	WY10200_00 AT  %MX10200.0 : BOOL; (*STN 5 PROCESS TANK HEATER A ON/OFF (-70K1) *)
	WY10200_01 AT  %MX10200.1 : BOOL; (*STN 5 PROCESS TANK HEATER A ON/OFF (-70K1) *)
	WY10200_02 AT  %MX10200.2 : BOOL; (*STN 5 PROCESS TANK HEATER A ON/OFF (-70K1) *)
	WY10200_03 AT  %MX10200.3 : BOOL; (*STN 5 PROCESS TANK HEATER A ON/OFF (-70K1) *)
	WY10200_04 AT  %MX10200.4 : BOOL; (*STN 5 PROCESS TANK HEATER A ON/OFF (-70K1) *)
	WY10200_05 AT  %MX10200.5 : BOOL; (*STN 5 PROCESS TANK HEATER A ON/OFF (-70K1) *)
	WY10200_06 AT  %MX10200.6 : BOOL; (*STN 5 PROCESS TANK HEATER A ON/OFF (-70K1) *)
	WY10200_07 AT  %MX10200.7 : BOOL; (*STN 5 PROCESS TANK HEATER A ON/OFF (-70K1) *)
	WY10200_08 AT  %MX10200.8 : BOOL; (*STN 5 PROCESS TANK HEATER A ON/OFF (-70K1) *)
	WY10200_09 AT  %MX10200.9 : BOOL; (*STN 5 PROCESS TANK HEATER A ON/OFF (-70K1) *)
	WY10200_10 AT  %MX10200.10 : BOOL; (*STN 5 PROCESS TANK HEATER A ON/OFF (-70K1) *)
	WY10200_11 AT  %MX10200.11 : BOOL; (*STN 5 PROCESS TANK HEATER A ON/OFF (-70K1) *)
	WY10200_12 AT  %MX10200.12 : BOOL; (*STN 5 PROCESS TANK HEATER A ON/OFF (-70K1) *)
	WY10200_13 AT  %MX10200.13 : BOOL; (*STN 5 PROCESS TANK HEATER A ON/OFF (-70K1) *)
	WY10200_14 AT  %MX10200.14 : BOOL; (*STN 5 PROCESS TANK HEATER A ON/OFF (-70K1) *)
	WY10200_15 AT  %MX10200.15 : BOOL; (*STN 5 PROCESS TANK HEATER A ON/OFF (-70K1) *)
	WY10200_16 AT  %MX10200.16 : BOOL; (*STN 5 PROCESS TANK HEATER A ON/OFF (-70K1) *)
	WY10200_17 AT  %MX10200.17 : BOOL; (*STN 5 PROCESS TANK HEATER A ON/OFF (-70K1) *)
	WY10200_18 AT  %MX10200.18 : BOOL; (*STN 5 PROCESS TANK HEATER A ON/OFF (-70K1) *)
	WY10200_19 AT  %MX10200.19 : BOOL; (*STN 5 PROCESS TANK HEATER A ON/OFF (-70K1) *)
	WY10200_20 AT  %MX10200.20 : BOOL; (*STN 5 PROCESS TANK HEATER A ON/OFF (-70K1) *)
	WY10200_21 AT  %MX10200.21 : BOOL; (*STN 5 PROCESS TANK HEATER A ON/OFF (-70K1) *)
	WY10200_22 AT  %MX10200.22 : BOOL; (*STN 5 PROCESS TANK HEATER A ON/OFF (-70K1) *)
	WY10200_23 AT  %MX10200.23 : BOOL; (*STN 5 PROCESS TANK HEATER A ON/OFF (-70K1) *)
	WY10200_24 AT  %MX10200.24 : BOOL; (*STN 5 PROCESS TANK HEATER A ON/OFF (-70K1) *)
	WY10200_25 AT  %MX10200.25 : BOOL; (*STN 5 PROCESS TANK HEATER A ON/OFF (-70K1) *)
	WY10200_26 AT  %MX10200.26 : BOOL; (*STN 5 PROCESS TANK HEATER A ON/OFF (-70K1) *)
	WY10200_27 AT  %MX10200.27 : BOOL; (*STN 5 PROCESS TANK HEATER A ON/OFF (-70K1) *)
	WY10200_28 AT  %MX10200.28 : BOOL; (*STN 5 PROCESS TANK HEATER A ON/OFF (-70K1) *)
	WY10200_29 AT  %MX10200.29 : BOOL; (*STN 5 PROCESS TANK HEATER A ON/OFF (-70K1) *)
	WY10200_30 AT  %MX10200.30 : BOOL; (*STN 5 PROCESS TANK HEATER A ON/OFF (-70K1) *)
	WY10200_31 AT  %MX10200.31 : BOOL; (*STN 5 PROCESS TANK HEATER A ON/OFF (-70K1) *)

	WY10201_00 AT  %MX10204.0 : BOOL; (*STN 5 PROCESS TANK HEATER B ON/OFF (-71K1) *)
	WY10201_01 AT  %MX10204.1 : BOOL; (*STN 5 PROCESS TANK HEATER B ON/OFF (-71K1) *)
	WY10201_02 AT  %MX10204.2 : BOOL; (*STN 5 PROCESS TANK HEATER B ON/OFF (-71K1) *)
	WY10201_03 AT  %MX10204.3 : BOOL; (*STN 5 PROCESS TANK HEATER B ON/OFF (-71K1) *)
	WY10201_04 AT  %MX10204.4 : BOOL; (*STN 5 PROCESS TANK HEATER B ON/OFF (-71K1) *)
	WY10201_05 AT  %MX10204.5 : BOOL; (*STN 5 PROCESS TANK HEATER B ON/OFF (-71K1) *)
	WY10201_06 AT  %MX10204.6 : BOOL; (*STN 5 PROCESS TANK HEATER B ON/OFF (-71K1) *)
	WY10201_07 AT  %MX10204.7 : BOOL; (*STN 5 PROCESS TANK HEATER B ON/OFF (-71K1) *)
	WY10201_08 AT  %MX10204.8 : BOOL; (*STN 5 PROCESS TANK HEATER B ON/OFF (-71K1) *)
	WY10201_09 AT  %MX10204.9 : BOOL; (*STN 5 PROCESS TANK HEATER B ON/OFF (-71K1) *)
	WY10201_10 AT  %MX10204.10 : BOOL; (*STN 5 PROCESS TANK HEATER B ON/OFF (-71K1) *)
	WY10201_11 AT  %MX10204.11 : BOOL; (*STN 5 PROCESS TANK HEATER B ON/OFF (-71K1) *)
	WY10201_12 AT  %MX10204.12 : BOOL; (*STN 5 PROCESS TANK HEATER B ON/OFF (-71K1) *)
	WY10201_13 AT  %MX10204.13 : BOOL; (*STN 5 PROCESS TANK HEATER B ON/OFF (-71K1) *)
	WY10201_14 AT  %MX10204.14 : BOOL; (*STN 5 PROCESS TANK HEATER B ON/OFF (-71K1) *)
	WY10201_15 AT  %MX10204.15 : BOOL; (*STN 5 PROCESS TANK HEATER B ON/OFF (-71K1) *)
	WY10201_16 AT  %MX10204.16 : BOOL; (*STN 5 PROCESS TANK HEATER B ON/OFF (-71K1) *)
	WY10201_17 AT  %MX10204.17 : BOOL; (*STN 5 PROCESS TANK HEATER B ON/OFF (-71K1) *)
	WY10201_18 AT  %MX10204.18 : BOOL; (*STN 5 PROCESS TANK HEATER B ON/OFF (-71K1) *)
	WY10201_19 AT  %MX10204.19 : BOOL; (*STN 5 PROCESS TANK HEATER B ON/OFF (-71K1) *)
	WY10201_20 AT  %MX10204.20 : BOOL; (*STN 5 PROCESS TANK HEATER B ON/OFF (-71K1) *)
	WY10201_21 AT  %MX10204.21 : BOOL; (*STN 5 PROCESS TANK HEATER B ON/OFF (-71K1) *)
	WY10201_22 AT  %MX10204.22 : BOOL; (*STN 5 PROCESS TANK HEATER B ON/OFF (-71K1) *)
	WY10201_23 AT  %MX10204.23 : BOOL; (*STN 5 PROCESS TANK HEATER B ON/OFF (-71K1) *)
	WY10201_24 AT  %MX10204.24 : BOOL; (*STN 5 PROCESS TANK HEATER B ON/OFF (-71K1) *)
	WY10201_25 AT  %MX10204.25 : BOOL; (*STN 5 PROCESS TANK HEATER B ON/OFF (-71K1) *)
	WY10201_26 AT  %MX10204.26 : BOOL; (*STN 5 PROCESS TANK HEATER B ON/OFF (-71K1) *)
	WY10201_27 AT  %MX10204.27 : BOOL; (*STN 5 PROCESS TANK HEATER B ON/OFF (-71K1) *)
	WY10201_28 AT  %MX10204.28 : BOOL; (*STN 5 PROCESS TANK HEATER B ON/OFF (-71K1) *)
	WY10201_29 AT  %MX10204.29 : BOOL; (*STN 5 PROCESS TANK HEATER B ON/OFF (-71K1) *)
	WY10201_30 AT  %MX10204.30 : BOOL; (*STN 5 PROCESS TANK HEATER B ON/OFF (-71K1) *)
	WY10201_31 AT  %MX10204.31 : BOOL; (*STN 5 PROCESS TANK HEATER B ON/OFF (-71K1) *)

	WY10202_00 AT  %MX10208.0 : BOOL; (*STN 1 SUB PROCESS TANK HEATER ON/OFF (-72K1) *)
	WY10202_01 AT  %MX10208.1 : BOOL; (*STN 1 SUB PROCESS TANK HEATER ON/OFF (-72K1) *)
	WY10202_02 AT  %MX10208.2 : BOOL; (*STN 1 SUB PROCESS TANK HEATER ON/OFF (-72K1) *)
	WY10202_03 AT  %MX10208.3 : BOOL; (*STN 1 SUB PROCESS TANK HEATER ON/OFF (-72K1) *)
	WY10202_04 AT  %MX10208.4 : BOOL; (*STN 1 SUB PROCESS TANK HEATER ON/OFF (-72K1) *)
	WY10202_05 AT  %MX10208.5 : BOOL; (*STN 1 SUB PROCESS TANK HEATER ON/OFF (-72K1) *)
	WY10202_06 AT  %MX10208.6 : BOOL; (*STN 1 SUB PROCESS TANK HEATER ON/OFF (-72K1) *)
	WY10202_07 AT  %MX10208.7 : BOOL; (*STN 1 SUB PROCESS TANK HEATER ON/OFF (-72K1) *)
	WY10202_08 AT  %MX10208.8 : BOOL; (*STN 1 SUB PROCESS TANK HEATER ON/OFF (-72K1) *)
	WY10202_09 AT  %MX10208.9 : BOOL; (*STN 1 SUB PROCESS TANK HEATER ON/OFF (-72K1) *)
	WY10202_10 AT  %MX10208.10 : BOOL; (*STN 1 SUB PROCESS TANK HEATER ON/OFF (-72K1) *)
	WY10202_11 AT  %MX10208.11 : BOOL; (*STN 1 SUB PROCESS TANK HEATER ON/OFF (-72K1) *)
	WY10202_12 AT  %MX10208.12 : BOOL; (*STN 1 SUB PROCESS TANK HEATER ON/OFF (-72K1) *)
	WY10202_13 AT  %MX10208.13 : BOOL; (*STN 1 SUB PROCESS TANK HEATER ON/OFF (-72K1) *)
	WY10202_14 AT  %MX10208.14 : BOOL; (*STN 1 SUB PROCESS TANK HEATER ON/OFF (-72K1) *)
	WY10202_15 AT  %MX10208.15 : BOOL; (*STN 1 SUB PROCESS TANK HEATER ON/OFF (-72K1) *)
	WY10202_16 AT  %MX10208.16 : BOOL; (*STN 1 SUB PROCESS TANK HEATER ON/OFF (-72K1) *)
	WY10202_17 AT  %MX10208.17 : BOOL; (*STN 1 SUB PROCESS TANK HEATER ON/OFF (-72K1) *)
	WY10202_18 AT  %MX10208.18 : BOOL; (*STN 1 SUB PROCESS TANK HEATER ON/OFF (-72K1) *)
	WY10202_19 AT  %MX10208.19 : BOOL; (*STN 1 SUB PROCESS TANK HEATER ON/OFF (-72K1) *)
	WY10202_20 AT  %MX10208.20 : BOOL; (*STN 1 SUB PROCESS TANK HEATER ON/OFF (-72K1) *)
	WY10202_21 AT  %MX10208.21 : BOOL; (*STN 1 SUB PROCESS TANK HEATER ON/OFF (-72K1) *)
	WY10202_22 AT  %MX10208.22 : BOOL; (*STN 1 SUB PROCESS TANK HEATER ON/OFF (-72K1) *)
	WY10202_23 AT  %MX10208.23 : BOOL; (*STN 1 SUB PROCESS TANK HEATER ON/OFF (-72K1) *)
	WY10202_24 AT  %MX10208.24 : BOOL; (*STN 1 SUB PROCESS TANK HEATER ON/OFF (-72K1) *)
	WY10202_25 AT  %MX10208.25 : BOOL; (*STN 1 SUB PROCESS TANK HEATER ON/OFF (-72K1) *)
	WY10202_26 AT  %MX10208.26 : BOOL; (*STN 1 SUB PROCESS TANK HEATER ON/OFF (-72K1) *)
	WY10202_27 AT  %MX10208.27 : BOOL; (*STN 1 SUB PROCESS TANK HEATER ON/OFF (-72K1) *)
	WY10202_28 AT  %MX10208.28 : BOOL; (*STN 1 SUB PROCESS TANK HEATER ON/OFF (-72K1) *)
	WY10202_29 AT  %MX10208.29 : BOOL; (*STN 1 SUB PROCESS TANK HEATER ON/OFF (-72K1) *)
	WY10202_30 AT  %MX10208.30 : BOOL; (*STN 1 SUB PROCESS TANK HEATER ON/OFF (-72K1) *)
	WY10202_31 AT  %MX10208.31 : BOOL; (*STN 1 SUB PROCESS TANK HEATER ON/OFF (-72K1) *)

	WY10203_00 AT  %MX10212.0 : BOOL; (*STN 2 SUB PROCESS TANK HEATER ON/OFF (-73K1) *)
	WY10203_01 AT  %MX10212.1 : BOOL; (*STN 2 SUB PROCESS TANK HEATER ON/OFF (-73K1) *)
	WY10203_02 AT  %MX10212.2 : BOOL; (*STN 2 SUB PROCESS TANK HEATER ON/OFF (-73K1) *)
	WY10203_03 AT  %MX10212.3 : BOOL; (*STN 2 SUB PROCESS TANK HEATER ON/OFF (-73K1) *)
	WY10203_04 AT  %MX10212.4 : BOOL; (*STN 2 SUB PROCESS TANK HEATER ON/OFF (-73K1) *)
	WY10203_05 AT  %MX10212.5 : BOOL; (*STN 2 SUB PROCESS TANK HEATER ON/OFF (-73K1) *)
	WY10203_06 AT  %MX10212.6 : BOOL; (*STN 2 SUB PROCESS TANK HEATER ON/OFF (-73K1) *)
	WY10203_07 AT  %MX10212.7 : BOOL; (*STN 2 SUB PROCESS TANK HEATER ON/OFF (-73K1) *)
	WY10203_08 AT  %MX10212.8 : BOOL; (*STN 2 SUB PROCESS TANK HEATER ON/OFF (-73K1) *)
	WY10203_09 AT  %MX10212.9 : BOOL; (*STN 2 SUB PROCESS TANK HEATER ON/OFF (-73K1) *)
	WY10203_10 AT  %MX10212.10 : BOOL; (*STN 2 SUB PROCESS TANK HEATER ON/OFF (-73K1) *)
	WY10203_11 AT  %MX10212.11 : BOOL; (*STN 2 SUB PROCESS TANK HEATER ON/OFF (-73K1) *)
	WY10203_12 AT  %MX10212.12 : BOOL; (*STN 2 SUB PROCESS TANK HEATER ON/OFF (-73K1) *)
	WY10203_13 AT  %MX10212.13 : BOOL; (*STN 2 SUB PROCESS TANK HEATER ON/OFF (-73K1) *)
	WY10203_14 AT  %MX10212.14 : BOOL; (*STN 2 SUB PROCESS TANK HEATER ON/OFF (-73K1) *)
	WY10203_15 AT  %MX10212.15 : BOOL; (*STN 2 SUB PROCESS TANK HEATER ON/OFF (-73K1) *)
	WY10203_16 AT  %MX10212.16 : BOOL; (*STN 2 SUB PROCESS TANK HEATER ON/OFF (-73K1) *)
	WY10203_17 AT  %MX10212.17 : BOOL; (*STN 2 SUB PROCESS TANK HEATER ON/OFF (-73K1) *)
	WY10203_18 AT  %MX10212.18 : BOOL; (*STN 2 SUB PROCESS TANK HEATER ON/OFF (-73K1) *)
	WY10203_19 AT  %MX10212.19 : BOOL; (*STN 2 SUB PROCESS TANK HEATER ON/OFF (-73K1) *)
	WY10203_20 AT  %MX10212.20 : BOOL; (*STN 2 SUB PROCESS TANK HEATER ON/OFF (-73K1) *)
	WY10203_21 AT  %MX10212.21 : BOOL; (*STN 2 SUB PROCESS TANK HEATER ON/OFF (-73K1) *)
	WY10203_22 AT  %MX10212.22 : BOOL; (*STN 2 SUB PROCESS TANK HEATER ON/OFF (-73K1) *)
	WY10203_23 AT  %MX10212.23 : BOOL; (*STN 2 SUB PROCESS TANK HEATER ON/OFF (-73K1) *)
	WY10203_24 AT  %MX10212.24 : BOOL; (*STN 2 SUB PROCESS TANK HEATER ON/OFF (-73K1) *)
	WY10203_25 AT  %MX10212.25 : BOOL; (*STN 2 SUB PROCESS TANK HEATER ON/OFF (-73K1) *)
	WY10203_26 AT  %MX10212.26 : BOOL; (*STN 2 SUB PROCESS TANK HEATER ON/OFF (-73K1) *)
	WY10203_27 AT  %MX10212.27 : BOOL; (*STN 2 SUB PROCESS TANK HEATER ON/OFF (-73K1) *)
	WY10203_28 AT  %MX10212.28 : BOOL; (*STN 2 SUB PROCESS TANK HEATER ON/OFF (-73K1) *)
	WY10203_29 AT  %MX10212.29 : BOOL; (*STN 2 SUB PROCESS TANK HEATER ON/OFF (-73K1) *)
	WY10203_30 AT  %MX10212.30 : BOOL; (*STN 2 SUB PROCESS TANK HEATER ON/OFF (-73K1) *)
	WY10203_31 AT  %MX10212.31 : BOOL; (*STN 2 SUB PROCESS TANK HEATER ON/OFF (-73K1) *)

	WY10204_00 AT  %MX10216.0 : BOOL; (*STN 3 SUB PROCESS TANK HEATER ON/OFF (-74K1) *)
	WY10204_01 AT  %MX10216.1 : BOOL; (*STN 3 SUB PROCESS TANK HEATER ON/OFF (-74K1) *)
	WY10204_02 AT  %MX10216.2 : BOOL; (*STN 3 SUB PROCESS TANK HEATER ON/OFF (-74K1) *)
	WY10204_03 AT  %MX10216.3 : BOOL; (*STN 3 SUB PROCESS TANK HEATER ON/OFF (-74K1) *)
	WY10204_04 AT  %MX10216.4 : BOOL; (*STN 3 SUB PROCESS TANK HEATER ON/OFF (-74K1) *)
	WY10204_05 AT  %MX10216.5 : BOOL; (*STN 3 SUB PROCESS TANK HEATER ON/OFF (-74K1) *)
	WY10204_06 AT  %MX10216.6 : BOOL; (*STN 3 SUB PROCESS TANK HEATER ON/OFF (-74K1) *)
	WY10204_07 AT  %MX10216.7 : BOOL; (*STN 3 SUB PROCESS TANK HEATER ON/OFF (-74K1) *)
	WY10204_08 AT  %MX10216.8 : BOOL; (*STN 3 SUB PROCESS TANK HEATER ON/OFF (-74K1) *)
	WY10204_09 AT  %MX10216.9 : BOOL; (*STN 3 SUB PROCESS TANK HEATER ON/OFF (-74K1) *)
	WY10204_10 AT  %MX10216.10 : BOOL; (*STN 3 SUB PROCESS TANK HEATER ON/OFF (-74K1) *)
	WY10204_11 AT  %MX10216.11 : BOOL; (*STN 3 SUB PROCESS TANK HEATER ON/OFF (-74K1) *)
	WY10204_12 AT  %MX10216.12 : BOOL; (*STN 3 SUB PROCESS TANK HEATER ON/OFF (-74K1) *)
	WY10204_13 AT  %MX10216.13 : BOOL; (*STN 3 SUB PROCESS TANK HEATER ON/OFF (-74K1) *)
	WY10204_14 AT  %MX10216.14 : BOOL; (*STN 3 SUB PROCESS TANK HEATER ON/OFF (-74K1) *)
	WY10204_15 AT  %MX10216.15 : BOOL; (*STN 3 SUB PROCESS TANK HEATER ON/OFF (-74K1) *)
	WY10204_16 AT  %MX10216.16 : BOOL; (*STN 3 SUB PROCESS TANK HEATER ON/OFF (-74K1) *)
	WY10204_17 AT  %MX10216.17 : BOOL; (*STN 3 SUB PROCESS TANK HEATER ON/OFF (-74K1) *)
	WY10204_18 AT  %MX10216.18 : BOOL; (*STN 3 SUB PROCESS TANK HEATER ON/OFF (-74K1) *)
	WY10204_19 AT  %MX10216.19 : BOOL; (*STN 3 SUB PROCESS TANK HEATER ON/OFF (-74K1) *)
	WY10204_20 AT  %MX10216.20 : BOOL; (*STN 3 SUB PROCESS TANK HEATER ON/OFF (-74K1) *)
	WY10204_21 AT  %MX10216.21 : BOOL; (*STN 3 SUB PROCESS TANK HEATER ON/OFF (-74K1) *)
	WY10204_22 AT  %MX10216.22 : BOOL; (*STN 3 SUB PROCESS TANK HEATER ON/OFF (-74K1) *)
	WY10204_23 AT  %MX10216.23 : BOOL; (*STN 3 SUB PROCESS TANK HEATER ON/OFF (-74K1) *)
	WY10204_24 AT  %MX10216.24 : BOOL; (*STN 3 SUB PROCESS TANK HEATER ON/OFF (-74K1) *)
	WY10204_25 AT  %MX10216.25 : BOOL; (*STN 3 SUB PROCESS TANK HEATER ON/OFF (-74K1) *)
	WY10204_26 AT  %MX10216.26 : BOOL; (*STN 3 SUB PROCESS TANK HEATER ON/OFF (-74K1) *)
	WY10204_27 AT  %MX10216.27 : BOOL; (*STN 3 SUB PROCESS TANK HEATER ON/OFF (-74K1) *)
	WY10204_28 AT  %MX10216.28 : BOOL; (*STN 3 SUB PROCESS TANK HEATER ON/OFF (-74K1) *)
	WY10204_29 AT  %MX10216.29 : BOOL; (*STN 3 SUB PROCESS TANK HEATER ON/OFF (-74K1) *)
	WY10204_30 AT  %MX10216.30 : BOOL; (*STN 3 SUB PROCESS TANK HEATER ON/OFF (-74K1) *)
	WY10204_31 AT  %MX10216.31 : BOOL; (*STN 3 SUB PROCESS TANK HEATER ON/OFF (-74K1) *)

	WY10205_00 AT  %MX10220.0 : BOOL; (*MAIN INC HEATER ON/OFF   (-75K1) *)
	WY10205_01 AT  %MX10220.1 : BOOL; (*MAIN INC HEATER ON/OFF   (-75K1) *)
	WY10205_02 AT  %MX10220.2 : BOOL; (*MAIN INC HEATER ON/OFF   (-75K1) *)
	WY10205_03 AT  %MX10220.3 : BOOL; (*MAIN INC HEATER ON/OFF   (-75K1) *)
	WY10205_04 AT  %MX10220.4 : BOOL; (*MAIN INC HEATER ON/OFF   (-75K1) *)
	WY10205_05 AT  %MX10220.5 : BOOL; (*MAIN INC HEATER ON/OFF   (-75K1) *)
	WY10205_06 AT  %MX10220.6 : BOOL; (*MAIN INC HEATER ON/OFF   (-75K1) *)
	WY10205_07 AT  %MX10220.7 : BOOL; (*MAIN INC HEATER ON/OFF   (-75K1) *)
	WY10205_08 AT  %MX10220.8 : BOOL; (*MAIN INC HEATER ON/OFF   (-75K1) *)
	WY10205_09 AT  %MX10220.9 : BOOL; (*MAIN INC HEATER ON/OFF   (-75K1) *)
	WY10205_10 AT  %MX10220.10 : BOOL; (*MAIN INC HEATER ON/OFF   (-75K1) *)
	WY10205_11 AT  %MX10220.11 : BOOL; (*MAIN INC HEATER ON/OFF   (-75K1) *)
	WY10205_12 AT  %MX10220.12 : BOOL; (*MAIN INC HEATER ON/OFF   (-75K1) *)
	WY10205_13 AT  %MX10220.13 : BOOL; (*MAIN INC HEATER ON/OFF   (-75K1) *)
	WY10205_14 AT  %MX10220.14 : BOOL; (*MAIN INC HEATER ON/OFF   (-75K1) *)
	WY10205_15 AT  %MX10220.15 : BOOL; (*MAIN INC HEATER ON/OFF   (-75K1) *)
	WY10205_16 AT  %MX10220.16 : BOOL; (*MAIN INC HEATER ON/OFF   (-75K1) *)
	WY10205_17 AT  %MX10220.17 : BOOL; (*MAIN INC HEATER ON/OFF   (-75K1) *)
	WY10205_18 AT  %MX10220.18 : BOOL; (*MAIN INC HEATER ON/OFF   (-75K1) *)
	WY10205_19 AT  %MX10220.19 : BOOL; (*MAIN INC HEATER ON/OFF   (-75K1) *)
	WY10205_20 AT  %MX10220.20 : BOOL; (*MAIN INC HEATER ON/OFF   (-75K1) *)
	WY10205_21 AT  %MX10220.21 : BOOL; (*MAIN INC HEATER ON/OFF   (-75K1) *)
	WY10205_22 AT  %MX10220.22 : BOOL; (*MAIN INC HEATER ON/OFF   (-75K1) *)
	WY10205_23 AT  %MX10220.23 : BOOL; (*MAIN INC HEATER ON/OFF   (-75K1) *)
	WY10205_24 AT  %MX10220.24 : BOOL; (*MAIN INC HEATER ON/OFF   (-75K1) *)
	WY10205_25 AT  %MX10220.25 : BOOL; (*MAIN INC HEATER ON/OFF   (-75K1) *)
	WY10205_26 AT  %MX10220.26 : BOOL; (*MAIN INC HEATER ON/OFF   (-75K1) *)
	WY10205_27 AT  %MX10220.27 : BOOL; (*MAIN INC HEATER ON/OFF   (-75K1) *)
	WY10205_28 AT  %MX10220.28 : BOOL; (*MAIN INC HEATER ON/OFF   (-75K1) *)
	WY10205_29 AT  %MX10220.29 : BOOL; (*MAIN INC HEATER ON/OFF   (-75K1) *)
	WY10205_30 AT  %MX10220.30 : BOOL; (*MAIN INC HEATER ON/OFF   (-75K1) *)
	WY10205_31 AT  %MX10220.31 : BOOL; (*MAIN INC HEATER ON/OFF   (-75K1) *)

	WY10206_00 AT  %MX10224.0 : BOOL; (*STN 1 ULTRASONIC FREQ ON/OFF (-16U1) *)
	WY10206_01 AT  %MX10224.1 : BOOL; (*STN 1 ULTRASONIC FREQ ON/OFF (-16U1) *)
	WY10206_02 AT  %MX10224.2 : BOOL; (*STN 1 ULTRASONIC FREQ ON/OFF (-16U1) *)
	WY10206_03 AT  %MX10224.3 : BOOL; (*STN 1 ULTRASONIC FREQ ON/OFF (-16U1) *)
	WY10206_04 AT  %MX10224.4 : BOOL; (*STN 1 ULTRASONIC FREQ ON/OFF (-16U1) *)
	WY10206_05 AT  %MX10224.5 : BOOL; (*STN 1 ULTRASONIC FREQ ON/OFF (-16U1) *)
	WY10206_06 AT  %MX10224.6 : BOOL; (*STN 1 ULTRASONIC FREQ ON/OFF (-16U1) *)
	WY10206_07 AT  %MX10224.7 : BOOL; (*STN 1 ULTRASONIC FREQ ON/OFF (-16U1) *)
	WY10206_08 AT  %MX10224.8 : BOOL; (*STN 1 ULTRASONIC FREQ ON/OFF (-16U1) *)
	WY10206_09 AT  %MX10224.9 : BOOL; (*STN 1 ULTRASONIC FREQ ON/OFF (-16U1) *)
	WY10206_10 AT  %MX10224.10 : BOOL; (*STN 1 ULTRASONIC FREQ ON/OFF (-16U1) *)
	WY10206_11 AT  %MX10224.11 : BOOL; (*STN 1 ULTRASONIC FREQ ON/OFF (-16U1) *)
	WY10206_12 AT  %MX10224.12 : BOOL; (*STN 1 ULTRASONIC FREQ ON/OFF (-16U1) *)
	WY10206_13 AT  %MX10224.13 : BOOL; (*STN 1 ULTRASONIC FREQ ON/OFF (-16U1) *)
	WY10206_14 AT  %MX10224.14 : BOOL; (*STN 1 ULTRASONIC FREQ ON/OFF (-16U1) *)
	WY10206_15 AT  %MX10224.15 : BOOL; (*STN 1 ULTRASONIC FREQ ON/OFF (-16U1) *)
	WY10206_16 AT  %MX10224.16 : BOOL; (*STN 1 ULTRASONIC FREQ ON/OFF (-16U1) *)
	WY10206_17 AT  %MX10224.17 : BOOL; (*STN 1 ULTRASONIC FREQ ON/OFF (-16U1) *)
	WY10206_18 AT  %MX10224.18 : BOOL; (*STN 1 ULTRASONIC FREQ ON/OFF (-16U1) *)
	WY10206_19 AT  %MX10224.19 : BOOL; (*STN 1 ULTRASONIC FREQ ON/OFF (-16U1) *)
	WY10206_20 AT  %MX10224.20 : BOOL; (*STN 1 ULTRASONIC FREQ ON/OFF (-16U1) *)
	WY10206_21 AT  %MX10224.21 : BOOL; (*STN 1 ULTRASONIC FREQ ON/OFF (-16U1) *)
	WY10206_22 AT  %MX10224.22 : BOOL; (*STN 1 ULTRASONIC FREQ ON/OFF (-16U1) *)
	WY10206_23 AT  %MX10224.23 : BOOL; (*STN 1 ULTRASONIC FREQ ON/OFF (-16U1) *)
	WY10206_24 AT  %MX10224.24 : BOOL; (*STN 1 ULTRASONIC FREQ ON/OFF (-16U1) *)
	WY10206_25 AT  %MX10224.25 : BOOL; (*STN 1 ULTRASONIC FREQ ON/OFF (-16U1) *)
	WY10206_26 AT  %MX10224.26 : BOOL; (*STN 1 ULTRASONIC FREQ ON/OFF (-16U1) *)
	WY10206_27 AT  %MX10224.27 : BOOL; (*STN 1 ULTRASONIC FREQ ON/OFF (-16U1) *)
	WY10206_28 AT  %MX10224.28 : BOOL; (*STN 1 ULTRASONIC FREQ ON/OFF (-16U1) *)
	WY10206_29 AT  %MX10224.29 : BOOL; (*STN 1 ULTRASONIC FREQ ON/OFF (-16U1) *)
	WY10206_30 AT  %MX10224.30 : BOOL; (*STN 1 ULTRASONIC FREQ ON/OFF (-16U1) *)
	WY10206_31 AT  %MX10224.31 : BOOL; (*STN 1 ULTRASONIC FREQ ON/OFF (-16U1) *)

	WY10207_00 AT  %MX10228.0 : BOOL; (*STN 2 ULTRASONIC FREQ ON/OFF (-17U1) *)
	WY10207_01 AT  %MX10228.1 : BOOL; (*STN 2 ULTRASONIC FREQ ON/OFF (-17U1) *)
	WY10207_02 AT  %MX10228.2 : BOOL; (*STN 2 ULTRASONIC FREQ ON/OFF (-17U1) *)
	WY10207_03 AT  %MX10228.3 : BOOL; (*STN 2 ULTRASONIC FREQ ON/OFF (-17U1) *)
	WY10207_04 AT  %MX10228.4 : BOOL; (*STN 2 ULTRASONIC FREQ ON/OFF (-17U1) *)
	WY10207_05 AT  %MX10228.5 : BOOL; (*STN 2 ULTRASONIC FREQ ON/OFF (-17U1) *)
	WY10207_06 AT  %MX10228.6 : BOOL; (*STN 2 ULTRASONIC FREQ ON/OFF (-17U1) *)
	WY10207_07 AT  %MX10228.7 : BOOL; (*STN 2 ULTRASONIC FREQ ON/OFF (-17U1) *)
	WY10207_08 AT  %MX10228.8 : BOOL; (*STN 2 ULTRASONIC FREQ ON/OFF (-17U1) *)
	WY10207_09 AT  %MX10228.9 : BOOL; (*STN 2 ULTRASONIC FREQ ON/OFF (-17U1) *)
	WY10207_10 AT  %MX10228.10 : BOOL; (*STN 2 ULTRASONIC FREQ ON/OFF (-17U1) *)
	WY10207_11 AT  %MX10228.11 : BOOL; (*STN 2 ULTRASONIC FREQ ON/OFF (-17U1) *)
	WY10207_12 AT  %MX10228.12 : BOOL; (*STN 2 ULTRASONIC FREQ ON/OFF (-17U1) *)
	WY10207_13 AT  %MX10228.13 : BOOL; (*STN 2 ULTRASONIC FREQ ON/OFF (-17U1) *)
	WY10207_14 AT  %MX10228.14 : BOOL; (*STN 2 ULTRASONIC FREQ ON/OFF (-17U1) *)
	WY10207_15 AT  %MX10228.15 : BOOL; (*STN 2 ULTRASONIC FREQ ON/OFF (-17U1) *)
	WY10207_16 AT  %MX10228.16 : BOOL; (*STN 2 ULTRASONIC FREQ ON/OFF (-17U1) *)
	WY10207_17 AT  %MX10228.17 : BOOL; (*STN 2 ULTRASONIC FREQ ON/OFF (-17U1) *)
	WY10207_18 AT  %MX10228.18 : BOOL; (*STN 2 ULTRASONIC FREQ ON/OFF (-17U1) *)
	WY10207_19 AT  %MX10228.19 : BOOL; (*STN 2 ULTRASONIC FREQ ON/OFF (-17U1) *)
	WY10207_20 AT  %MX10228.20 : BOOL; (*STN 2 ULTRASONIC FREQ ON/OFF (-17U1) *)
	WY10207_21 AT  %MX10228.21 : BOOL; (*STN 2 ULTRASONIC FREQ ON/OFF (-17U1) *)
	WY10207_22 AT  %MX10228.22 : BOOL; (*STN 2 ULTRASONIC FREQ ON/OFF (-17U1) *)
	WY10207_23 AT  %MX10228.23 : BOOL; (*STN 2 ULTRASONIC FREQ ON/OFF (-17U1) *)
	WY10207_24 AT  %MX10228.24 : BOOL; (*STN 2 ULTRASONIC FREQ ON/OFF (-17U1) *)
	WY10207_25 AT  %MX10228.25 : BOOL; (*STN 2 ULTRASONIC FREQ ON/OFF (-17U1) *)
	WY10207_26 AT  %MX10228.26 : BOOL; (*STN 2 ULTRASONIC FREQ ON/OFF (-17U1) *)
	WY10207_27 AT  %MX10228.27 : BOOL; (*STN 2 ULTRASONIC FREQ ON/OFF (-17U1) *)
	WY10207_28 AT  %MX10228.28 : BOOL; (*STN 2 ULTRASONIC FREQ ON/OFF (-17U1) *)
	WY10207_29 AT  %MX10228.29 : BOOL; (*STN 2 ULTRASONIC FREQ ON/OFF (-17U1) *)
	WY10207_30 AT  %MX10228.30 : BOOL; (*STN 2 ULTRASONIC FREQ ON/OFF (-17U1) *)
	WY10207_31 AT  %MX10228.31 : BOOL; (*STN 2 ULTRASONIC FREQ ON/OFF (-17U1) *)

	WY10208_00 AT  %MX10232.0 : BOOL; (*STN 3 ULTRASONIC FREQ ON/OFF (-18U1) *)
	WY10208_01 AT  %MX10232.1 : BOOL; (*STN 3 ULTRASONIC FREQ ON/OFF (-18U1) *)
	WY10208_02 AT  %MX10232.2 : BOOL; (*STN 3 ULTRASONIC FREQ ON/OFF (-18U1) *)
	WY10208_03 AT  %MX10232.3 : BOOL; (*STN 3 ULTRASONIC FREQ ON/OFF (-18U1) *)
	WY10208_04 AT  %MX10232.4 : BOOL; (*STN 3 ULTRASONIC FREQ ON/OFF (-18U1) *)
	WY10208_05 AT  %MX10232.5 : BOOL; (*STN 3 ULTRASONIC FREQ ON/OFF (-18U1) *)
	WY10208_06 AT  %MX10232.6 : BOOL; (*STN 3 ULTRASONIC FREQ ON/OFF (-18U1) *)
	WY10208_07 AT  %MX10232.7 : BOOL; (*STN 3 ULTRASONIC FREQ ON/OFF (-18U1) *)
	WY10208_08 AT  %MX10232.8 : BOOL; (*STN 3 ULTRASONIC FREQ ON/OFF (-18U1) *)
	WY10208_09 AT  %MX10232.9 : BOOL; (*STN 3 ULTRASONIC FREQ ON/OFF (-18U1) *)
	WY10208_10 AT  %MX10232.10 : BOOL; (*STN 3 ULTRASONIC FREQ ON/OFF (-18U1) *)
	WY10208_11 AT  %MX10232.11 : BOOL; (*STN 3 ULTRASONIC FREQ ON/OFF (-18U1) *)
	WY10208_12 AT  %MX10232.12 : BOOL; (*STN 3 ULTRASONIC FREQ ON/OFF (-18U1) *)
	WY10208_13 AT  %MX10232.13 : BOOL; (*STN 3 ULTRASONIC FREQ ON/OFF (-18U1) *)
	WY10208_14 AT  %MX10232.14 : BOOL; (*STN 3 ULTRASONIC FREQ ON/OFF (-18U1) *)
	WY10208_15 AT  %MX10232.15 : BOOL; (*STN 3 ULTRASONIC FREQ ON/OFF (-18U1) *)
	WY10208_16 AT  %MX10232.16 : BOOL; (*STN 3 ULTRASONIC FREQ ON/OFF (-18U1) *)
	WY10208_17 AT  %MX10232.17 : BOOL; (*STN 3 ULTRASONIC FREQ ON/OFF (-18U1) *)
	WY10208_18 AT  %MX10232.18 : BOOL; (*STN 3 ULTRASONIC FREQ ON/OFF (-18U1) *)
	WY10208_19 AT  %MX10232.19 : BOOL; (*STN 3 ULTRASONIC FREQ ON/OFF (-18U1) *)
	WY10208_20 AT  %MX10232.20 : BOOL; (*STN 3 ULTRASONIC FREQ ON/OFF (-18U1) *)
	WY10208_21 AT  %MX10232.21 : BOOL; (*STN 3 ULTRASONIC FREQ ON/OFF (-18U1) *)
	WY10208_22 AT  %MX10232.22 : BOOL; (*STN 3 ULTRASONIC FREQ ON/OFF (-18U1) *)
	WY10208_23 AT  %MX10232.23 : BOOL; (*STN 3 ULTRASONIC FREQ ON/OFF (-18U1) *)
	WY10208_24 AT  %MX10232.24 : BOOL; (*STN 3 ULTRASONIC FREQ ON/OFF (-18U1) *)
	WY10208_25 AT  %MX10232.25 : BOOL; (*STN 3 ULTRASONIC FREQ ON/OFF (-18U1) *)
	WY10208_26 AT  %MX10232.26 : BOOL; (*STN 3 ULTRASONIC FREQ ON/OFF (-18U1) *)
	WY10208_27 AT  %MX10232.27 : BOOL; (*STN 3 ULTRASONIC FREQ ON/OFF (-18U1) *)
	WY10208_28 AT  %MX10232.28 : BOOL; (*STN 3 ULTRASONIC FREQ ON/OFF (-18U1) *)
	WY10208_29 AT  %MX10232.29 : BOOL; (*STN 3 ULTRASONIC FREQ ON/OFF (-18U1) *)
	WY10208_30 AT  %MX10232.30 : BOOL; (*STN 3 ULTRASONIC FREQ ON/OFF (-18U1) *)
	WY10208_31 AT  %MX10232.31 : BOOL; (*STN 3 ULTRASONIC FREQ ON/OFF (-18U1) *)

	WY10209_00 AT  %MX10236.0 : BOOL; (*RESERVED *)
	WY10209_01 AT  %MX10236.1 : BOOL; (*RESERVED *)
	WY10209_02 AT  %MX10236.2 : BOOL; (*RESERVED *)
	WY10209_03 AT  %MX10236.3 : BOOL; (*RESERVED *)
	WY10209_04 AT  %MX10236.4 : BOOL; (*RESERVED *)
	WY10209_05 AT  %MX10236.5 : BOOL; (*RESERVED *)
	WY10209_06 AT  %MX10236.6 : BOOL; (*RESERVED *)
	WY10209_07 AT  %MX10236.7 : BOOL; (*RESERVED *)
	WY10209_08 AT  %MX10236.8 : BOOL; (*RESERVED *)
	WY10209_09 AT  %MX10236.9 : BOOL; (*RESERVED *)
	WY10209_10 AT  %MX10236.10 : BOOL; (*RESERVED *)
	WY10209_11 AT  %MX10236.11 : BOOL; (*RESERVED *)
	WY10209_12 AT  %MX10236.12 : BOOL; (*RESERVED *)
	WY10209_13 AT  %MX10236.13 : BOOL; (*RESERVED *)
	WY10209_14 AT  %MX10236.14 : BOOL; (*RESERVED *)
	WY10209_15 AT  %MX10236.15 : BOOL; (*RESERVED *)
	WY10209_16 AT  %MX10236.16 : BOOL; (*RESERVED *)
	WY10209_17 AT  %MX10236.17 : BOOL; (*RESERVED *)
	WY10209_18 AT  %MX10236.18 : BOOL; (*RESERVED *)
	WY10209_19 AT  %MX10236.19 : BOOL; (*RESERVED *)
	WY10209_20 AT  %MX10236.20 : BOOL; (*RESERVED *)
	WY10209_21 AT  %MX10236.21 : BOOL; (*RESERVED *)
	WY10209_22 AT  %MX10236.22 : BOOL; (*RESERVED *)
	WY10209_23 AT  %MX10236.23 : BOOL; (*RESERVED *)
	WY10209_24 AT  %MX10236.24 : BOOL; (*RESERVED *)
	WY10209_25 AT  %MX10236.25 : BOOL; (*RESERVED *)
	WY10209_26 AT  %MX10236.26 : BOOL; (*RESERVED *)
	WY10209_27 AT  %MX10236.27 : BOOL; (*RESERVED *)
	WY10209_28 AT  %MX10236.28 : BOOL; (*RESERVED *)
	WY10209_29 AT  %MX10236.29 : BOOL; (*RESERVED *)
	WY10209_30 AT  %MX10236.30 : BOOL; (*RESERVED *)
	WY10209_31 AT  %MX10236.31 : BOOL; (*RESERVED *)

	WY10210_00 AT  %MX10240.0 : BOOL; (*RESERVED *)
	WY10210_01 AT  %MX10240.1 : BOOL; (*RESERVED *)
	WY10210_02 AT  %MX10240.2 : BOOL; (*RESERVED *)
	WY10210_03 AT  %MX10240.3 : BOOL; (*RESERVED *)
	WY10210_04 AT  %MX10240.4 : BOOL; (*RESERVED *)
	WY10210_05 AT  %MX10240.5 : BOOL; (*RESERVED *)
	WY10210_06 AT  %MX10240.6 : BOOL; (*RESERVED *)
	WY10210_07 AT  %MX10240.7 : BOOL; (*RESERVED *)
	WY10210_08 AT  %MX10240.8 : BOOL; (*RESERVED *)
	WY10210_09 AT  %MX10240.9 : BOOL; (*RESERVED *)
	WY10210_10 AT  %MX10240.10 : BOOL; (*RESERVED *)
	WY10210_11 AT  %MX10240.11 : BOOL; (*RESERVED *)
	WY10210_12 AT  %MX10240.12 : BOOL; (*RESERVED *)
	WY10210_13 AT  %MX10240.13 : BOOL; (*RESERVED *)
	WY10210_14 AT  %MX10240.14 : BOOL; (*RESERVED *)
	WY10210_15 AT  %MX10240.15 : BOOL; (*RESERVED *)
	WY10210_16 AT  %MX10240.16 : BOOL; (*RESERVED *)
	WY10210_17 AT  %MX10240.17 : BOOL; (*RESERVED *)
	WY10210_18 AT  %MX10240.18 : BOOL; (*RESERVED *)
	WY10210_19 AT  %MX10240.19 : BOOL; (*RESERVED *)
	WY10210_20 AT  %MX10240.20 : BOOL; (*RESERVED *)
	WY10210_21 AT  %MX10240.21 : BOOL; (*RESERVED *)
	WY10210_22 AT  %MX10240.22 : BOOL; (*RESERVED *)
	WY10210_23 AT  %MX10240.23 : BOOL; (*RESERVED *)
	WY10210_24 AT  %MX10240.24 : BOOL; (*RESERVED *)
	WY10210_25 AT  %MX10240.25 : BOOL; (*RESERVED *)
	WY10210_26 AT  %MX10240.26 : BOOL; (*RESERVED *)
	WY10210_27 AT  %MX10240.27 : BOOL; (*RESERVED *)
	WY10210_28 AT  %MX10240.28 : BOOL; (*RESERVED *)
	WY10210_29 AT  %MX10240.29 : BOOL; (*RESERVED *)
	WY10210_30 AT  %MX10240.30 : BOOL; (*RESERVED *)
	WY10210_31 AT  %MX10240.31 : BOOL; (*RESERVED *)

	WY10211_00 AT  %MX10244.0 : BOOL; (*RESERVED *)
	WY10211_01 AT  %MX10244.1 : BOOL; (*RESERVED *)
	WY10211_02 AT  %MX10244.2 : BOOL; (*RESERVED *)
	WY10211_03 AT  %MX10244.3 : BOOL; (*RESERVED *)
	WY10211_04 AT  %MX10244.4 : BOOL; (*RESERVED *)
	WY10211_05 AT  %MX10244.5 : BOOL; (*RESERVED *)
	WY10211_06 AT  %MX10244.6 : BOOL; (*RESERVED *)
	WY10211_07 AT  %MX10244.7 : BOOL; (*RESERVED *)
	WY10211_08 AT  %MX10244.8 : BOOL; (*RESERVED *)
	WY10211_09 AT  %MX10244.9 : BOOL; (*RESERVED *)
	WY10211_10 AT  %MX10244.10 : BOOL; (*RESERVED *)
	WY10211_11 AT  %MX10244.11 : BOOL; (*RESERVED *)
	WY10211_12 AT  %MX10244.12 : BOOL; (*RESERVED *)
	WY10211_13 AT  %MX10244.13 : BOOL; (*RESERVED *)
	WY10211_14 AT  %MX10244.14 : BOOL; (*RESERVED *)
	WY10211_15 AT  %MX10244.15 : BOOL; (*RESERVED *)
	WY10211_16 AT  %MX10244.16 : BOOL; (*RESERVED *)
	WY10211_17 AT  %MX10244.17 : BOOL; (*RESERVED *)
	WY10211_18 AT  %MX10244.18 : BOOL; (*RESERVED *)
	WY10211_19 AT  %MX10244.19 : BOOL; (*RESERVED *)
	WY10211_20 AT  %MX10244.20 : BOOL; (*RESERVED *)
	WY10211_21 AT  %MX10244.21 : BOOL; (*RESERVED *)
	WY10211_22 AT  %MX10244.22 : BOOL; (*RESERVED *)
	WY10211_23 AT  %MX10244.23 : BOOL; (*RESERVED *)
	WY10211_24 AT  %MX10244.24 : BOOL; (*RESERVED *)
	WY10211_25 AT  %MX10244.25 : BOOL; (*RESERVED *)
	WY10211_26 AT  %MX10244.26 : BOOL; (*RESERVED *)
	WY10211_27 AT  %MX10244.27 : BOOL; (*RESERVED *)
	WY10211_28 AT  %MX10244.28 : BOOL; (*RESERVED *)
	WY10211_29 AT  %MX10244.29 : BOOL; (*RESERVED *)
	WY10211_30 AT  %MX10244.30 : BOOL; (*RESERVED *)
	WY10211_31 AT  %MX10244.31 : BOOL; (*RESERVED *)

	WY10212_00 AT  %MX10248.0 : BOOL; (*RESERVED *)
	WY10212_01 AT  %MX10248.1 : BOOL; (*RESERVED *)
	WY10212_02 AT  %MX10248.2 : BOOL; (*RESERVED *)
	WY10212_03 AT  %MX10248.3 : BOOL; (*RESERVED *)
	WY10212_04 AT  %MX10248.4 : BOOL; (*RESERVED *)
	WY10212_05 AT  %MX10248.5 : BOOL; (*RESERVED *)
	WY10212_06 AT  %MX10248.6 : BOOL; (*RESERVED *)
	WY10212_07 AT  %MX10248.7 : BOOL; (*RESERVED *)
	WY10212_08 AT  %MX10248.8 : BOOL; (*RESERVED *)
	WY10212_09 AT  %MX10248.9 : BOOL; (*RESERVED *)
	WY10212_10 AT  %MX10248.10 : BOOL; (*RESERVED *)
	WY10212_11 AT  %MX10248.11 : BOOL; (*RESERVED *)
	WY10212_12 AT  %MX10248.12 : BOOL; (*RESERVED *)
	WY10212_13 AT  %MX10248.13 : BOOL; (*RESERVED *)
	WY10212_14 AT  %MX10248.14 : BOOL; (*RESERVED *)
	WY10212_15 AT  %MX10248.15 : BOOL; (*RESERVED *)
	WY10212_16 AT  %MX10248.16 : BOOL; (*RESERVED *)
	WY10212_17 AT  %MX10248.17 : BOOL; (*RESERVED *)
	WY10212_18 AT  %MX10248.18 : BOOL; (*RESERVED *)
	WY10212_19 AT  %MX10248.19 : BOOL; (*RESERVED *)
	WY10212_20 AT  %MX10248.20 : BOOL; (*RESERVED *)
	WY10212_21 AT  %MX10248.21 : BOOL; (*RESERVED *)
	WY10212_22 AT  %MX10248.22 : BOOL; (*RESERVED *)
	WY10212_23 AT  %MX10248.23 : BOOL; (*RESERVED *)
	WY10212_24 AT  %MX10248.24 : BOOL; (*RESERVED *)
	WY10212_25 AT  %MX10248.25 : BOOL; (*RESERVED *)
	WY10212_26 AT  %MX10248.26 : BOOL; (*RESERVED *)
	WY10212_27 AT  %MX10248.27 : BOOL; (*RESERVED *)
	WY10212_28 AT  %MX10248.28 : BOOL; (*RESERVED *)
	WY10212_29 AT  %MX10248.29 : BOOL; (*RESERVED *)
	WY10212_30 AT  %MX10248.30 : BOOL; (*RESERVED *)
	WY10212_31 AT  %MX10248.31 : BOOL; (*RESERVED *)

	WY10213_00 AT  %MX10252.0 : BOOL; (*RESERVED *)
	WY10213_01 AT  %MX10252.1 : BOOL; (*RESERVED *)
	WY10213_02 AT  %MX10252.2 : BOOL; (*RESERVED *)
	WY10213_03 AT  %MX10252.3 : BOOL; (*RESERVED *)
	WY10213_04 AT  %MX10252.4 : BOOL; (*RESERVED *)
	WY10213_05 AT  %MX10252.5 : BOOL; (*RESERVED *)
	WY10213_06 AT  %MX10252.6 : BOOL; (*RESERVED *)
	WY10213_07 AT  %MX10252.7 : BOOL; (*RESERVED *)
	WY10213_08 AT  %MX10252.8 : BOOL; (*RESERVED *)
	WY10213_09 AT  %MX10252.9 : BOOL; (*RESERVED *)
	WY10213_10 AT  %MX10252.10 : BOOL; (*RESERVED *)
	WY10213_11 AT  %MX10252.11 : BOOL; (*RESERVED *)
	WY10213_12 AT  %MX10252.12 : BOOL; (*RESERVED *)
	WY10213_13 AT  %MX10252.13 : BOOL; (*RESERVED *)
	WY10213_14 AT  %MX10252.14 : BOOL; (*RESERVED *)
	WY10213_15 AT  %MX10252.15 : BOOL; (*RESERVED *)
	WY10213_16 AT  %MX10252.16 : BOOL; (*RESERVED *)
	WY10213_17 AT  %MX10252.17 : BOOL; (*RESERVED *)
	WY10213_18 AT  %MX10252.18 : BOOL; (*RESERVED *)
	WY10213_19 AT  %MX10252.19 : BOOL; (*RESERVED *)
	WY10213_20 AT  %MX10252.20 : BOOL; (*RESERVED *)
	WY10213_21 AT  %MX10252.21 : BOOL; (*RESERVED *)
	WY10213_22 AT  %MX10252.22 : BOOL; (*RESERVED *)
	WY10213_23 AT  %MX10252.23 : BOOL; (*RESERVED *)
	WY10213_24 AT  %MX10252.24 : BOOL; (*RESERVED *)
	WY10213_25 AT  %MX10252.25 : BOOL; (*RESERVED *)
	WY10213_26 AT  %MX10252.26 : BOOL; (*RESERVED *)
	WY10213_27 AT  %MX10252.27 : BOOL; (*RESERVED *)
	WY10213_28 AT  %MX10252.28 : BOOL; (*RESERVED *)
	WY10213_29 AT  %MX10252.29 : BOOL; (*RESERVED *)
	WY10213_30 AT  %MX10252.30 : BOOL; (*RESERVED *)
	WY10213_31 AT  %MX10252.31 : BOOL; (*RESERVED *)

	WY10214_00 AT  %MX10256.0 : BOOL; (*RESERVED *)
	WY10214_01 AT  %MX10256.1 : BOOL; (*RESERVED *)
	WY10214_02 AT  %MX10256.2 : BOOL; (*RESERVED *)
	WY10214_03 AT  %MX10256.3 : BOOL; (*RESERVED *)
	WY10214_04 AT  %MX10256.4 : BOOL; (*RESERVED *)
	WY10214_05 AT  %MX10256.5 : BOOL; (*RESERVED *)
	WY10214_06 AT  %MX10256.6 : BOOL; (*RESERVED *)
	WY10214_07 AT  %MX10256.7 : BOOL; (*RESERVED *)
	WY10214_08 AT  %MX10256.8 : BOOL; (*RESERVED *)
	WY10214_09 AT  %MX10256.9 : BOOL; (*RESERVED *)
	WY10214_10 AT  %MX10256.10 : BOOL; (*RESERVED *)
	WY10214_11 AT  %MX10256.11 : BOOL; (*RESERVED *)
	WY10214_12 AT  %MX10256.12 : BOOL; (*RESERVED *)
	WY10214_13 AT  %MX10256.13 : BOOL; (*RESERVED *)
	WY10214_14 AT  %MX10256.14 : BOOL; (*RESERVED *)
	WY10214_15 AT  %MX10256.15 : BOOL; (*RESERVED *)
	WY10214_16 AT  %MX10256.16 : BOOL; (*RESERVED *)
	WY10214_17 AT  %MX10256.17 : BOOL; (*RESERVED *)
	WY10214_18 AT  %MX10256.18 : BOOL; (*RESERVED *)
	WY10214_19 AT  %MX10256.19 : BOOL; (*RESERVED *)
	WY10214_20 AT  %MX10256.20 : BOOL; (*RESERVED *)
	WY10214_21 AT  %MX10256.21 : BOOL; (*RESERVED *)
	WY10214_22 AT  %MX10256.22 : BOOL; (*RESERVED *)
	WY10214_23 AT  %MX10256.23 : BOOL; (*RESERVED *)
	WY10214_24 AT  %MX10256.24 : BOOL; (*RESERVED *)
	WY10214_25 AT  %MX10256.25 : BOOL; (*RESERVED *)
	WY10214_26 AT  %MX10256.26 : BOOL; (*RESERVED *)
	WY10214_27 AT  %MX10256.27 : BOOL; (*RESERVED *)
	WY10214_28 AT  %MX10256.28 : BOOL; (*RESERVED *)
	WY10214_29 AT  %MX10256.29 : BOOL; (*RESERVED *)
	WY10214_30 AT  %MX10256.30 : BOOL; (*RESERVED *)
	WY10214_31 AT  %MX10256.31 : BOOL; (*RESERVED *)

	WY10215_00 AT  %MX10260.0 : BOOL; (*RESERVED *)
	WY10215_01 AT  %MX10260.1 : BOOL; (*RESERVED *)
	WY10215_02 AT  %MX10260.2 : BOOL; (*RESERVED *)
	WY10215_03 AT  %MX10260.3 : BOOL; (*RESERVED *)
	WY10215_04 AT  %MX10260.4 : BOOL; (*RESERVED *)
	WY10215_05 AT  %MX10260.5 : BOOL; (*RESERVED *)
	WY10215_06 AT  %MX10260.6 : BOOL; (*RESERVED *)
	WY10215_07 AT  %MX10260.7 : BOOL; (*RESERVED *)
	WY10215_08 AT  %MX10260.8 : BOOL; (*RESERVED *)
	WY10215_09 AT  %MX10260.9 : BOOL; (*RESERVED *)
	WY10215_10 AT  %MX10260.10 : BOOL; (*RESERVED *)
	WY10215_11 AT  %MX10260.11 : BOOL; (*RESERVED *)
	WY10215_12 AT  %MX10260.12 : BOOL; (*RESERVED *)
	WY10215_13 AT  %MX10260.13 : BOOL; (*RESERVED *)
	WY10215_14 AT  %MX10260.14 : BOOL; (*RESERVED *)
	WY10215_15 AT  %MX10260.15 : BOOL; (*RESERVED *)
	WY10215_16 AT  %MX10260.16 : BOOL; (*RESERVED *)
	WY10215_17 AT  %MX10260.17 : BOOL; (*RESERVED *)
	WY10215_18 AT  %MX10260.18 : BOOL; (*RESERVED *)
	WY10215_19 AT  %MX10260.19 : BOOL; (*RESERVED *)
	WY10215_20 AT  %MX10260.20 : BOOL; (*RESERVED *)
	WY10215_21 AT  %MX10260.21 : BOOL; (*RESERVED *)
	WY10215_22 AT  %MX10260.22 : BOOL; (*RESERVED *)
	WY10215_23 AT  %MX10260.23 : BOOL; (*RESERVED *)
	WY10215_24 AT  %MX10260.24 : BOOL; (*RESERVED *)
	WY10215_25 AT  %MX10260.25 : BOOL; (*RESERVED *)
	WY10215_26 AT  %MX10260.26 : BOOL; (*RESERVED *)
	WY10215_27 AT  %MX10260.27 : BOOL; (*RESERVED *)
	WY10215_28 AT  %MX10260.28 : BOOL; (*RESERVED *)
	WY10215_29 AT  %MX10260.29 : BOOL; (*RESERVED *)
	WY10215_30 AT  %MX10260.30 : BOOL; (*RESERVED *)
	WY10215_31 AT  %MX10260.31 : BOOL; (*RESERVED *)

	WY11500_00 AT  %MX11500.0 : BOOL; (*STN 1 SLIDING DOOR - OPEN (-160Y1) *)
	WY11500_01 AT  %MX11500.1 : BOOL; (*STN 1 SLIDING DOOR - OPEN (-160Y1) *)
	WY11500_02 AT  %MX11500.2 : BOOL; (*STN 1 SLIDING DOOR - OPEN (-160Y1) *)
	WY11500_03 AT  %MX11500.3 : BOOL; (*STN 1 SLIDING DOOR - OPEN (-160Y1) *)
	WY11500_04 AT  %MX11500.4 : BOOL; (*STN 1 SLIDING DOOR - OPEN (-160Y1) *)
	WY11500_05 AT  %MX11500.5 : BOOL; (*STN 1 SLIDING DOOR - OPEN (-160Y1) *)
	WY11500_06 AT  %MX11500.6 : BOOL; (*STN 1 SLIDING DOOR - OPEN (-160Y1) *)
	WY11500_07 AT  %MX11500.7 : BOOL; (*STN 1 SLIDING DOOR - OPEN (-160Y1) *)
	WY11500_08 AT  %MX11500.8 : BOOL; (*STN 1 SLIDING DOOR - OPEN (-160Y1) *)
	WY11500_09 AT  %MX11500.9 : BOOL; (*STN 1 SLIDING DOOR - OPEN (-160Y1) *)
	WY11500_10 AT  %MX11500.10 : BOOL; (*STN 1 SLIDING DOOR - OPEN (-160Y1) *)
	WY11500_11 AT  %MX11500.11 : BOOL; (*STN 1 SLIDING DOOR - OPEN (-160Y1) *)
	WY11500_12 AT  %MX11500.12 : BOOL; (*STN 1 SLIDING DOOR - OPEN (-160Y1) *)
	WY11500_13 AT  %MX11500.13 : BOOL; (*STN 1 SLIDING DOOR - OPEN (-160Y1) *)
	WY11500_14 AT  %MX11500.14 : BOOL; (*STN 1 SLIDING DOOR - OPEN (-160Y1) *)
	WY11500_15 AT  %MX11500.15 : BOOL; (*STN 1 SLIDING DOOR - OPEN (-160Y1) *)
	WY11500_16 AT  %MX11500.16 : BOOL; (*STN 1 SLIDING DOOR - OPEN (-160Y1) *)
	WY11500_17 AT  %MX11500.17 : BOOL; (*STN 1 SLIDING DOOR - OPEN (-160Y1) *)
	WY11500_18 AT  %MX11500.18 : BOOL; (*STN 1 SLIDING DOOR - OPEN (-160Y1) *)
	WY11500_19 AT  %MX11500.19 : BOOL; (*STN 1 SLIDING DOOR - OPEN (-160Y1) *)
	WY11500_20 AT  %MX11500.20 : BOOL; (*STN 1 SLIDING DOOR - OPEN (-160Y1) *)
	WY11500_21 AT  %MX11500.21 : BOOL; (*STN 1 SLIDING DOOR - OPEN (-160Y1) *)
	WY11500_22 AT  %MX11500.22 : BOOL; (*STN 1 SLIDING DOOR - OPEN (-160Y1) *)
	WY11500_23 AT  %MX11500.23 : BOOL; (*STN 1 SLIDING DOOR - OPEN (-160Y1) *)
	WY11500_24 AT  %MX11500.24 : BOOL; (*STN 1 SLIDING DOOR - OPEN (-160Y1) *)
	WY11500_25 AT  %MX11500.25 : BOOL; (*STN 1 SLIDING DOOR - OPEN (-160Y1) *)
	WY11500_26 AT  %MX11500.26 : BOOL; (*STN 1 SLIDING DOOR - OPEN (-160Y1) *)
	WY11500_27 AT  %MX11500.27 : BOOL; (*STN 1 SLIDING DOOR - OPEN (-160Y1) *)
	WY11500_28 AT  %MX11500.28 : BOOL; (*STN 1 SLIDING DOOR - OPEN (-160Y1) *)
	WY11500_29 AT  %MX11500.29 : BOOL; (*STN 1 SLIDING DOOR - OPEN (-160Y1) *)
	WY11500_30 AT  %MX11500.30 : BOOL; (*STN 1 SLIDING DOOR - OPEN (-160Y1) *)
	WY11500_31 AT  %MX11500.31 : BOOL; (*STN 1 SLIDING DOOR - OPEN (-160Y1) *)

	WY11501_00 AT  %MX11504.0 : BOOL; (*STN 1 SLIDING DOOR - CLOSE (-160Y2) *)
	WY11501_01 AT  %MX11504.1 : BOOL; (*STN 1 SLIDING DOOR - CLOSE (-160Y2) *)
	WY11501_02 AT  %MX11504.2 : BOOL; (*STN 1 SLIDING DOOR - CLOSE (-160Y2) *)
	WY11501_03 AT  %MX11504.3 : BOOL; (*STN 1 SLIDING DOOR - CLOSE (-160Y2) *)
	WY11501_04 AT  %MX11504.4 : BOOL; (*STN 1 SLIDING DOOR - CLOSE (-160Y2) *)
	WY11501_05 AT  %MX11504.5 : BOOL; (*STN 1 SLIDING DOOR - CLOSE (-160Y2) *)
	WY11501_06 AT  %MX11504.6 : BOOL; (*STN 1 SLIDING DOOR - CLOSE (-160Y2) *)
	WY11501_07 AT  %MX11504.7 : BOOL; (*STN 1 SLIDING DOOR - CLOSE (-160Y2) *)
	WY11501_08 AT  %MX11504.8 : BOOL; (*STN 1 SLIDING DOOR - CLOSE (-160Y2) *)
	WY11501_09 AT  %MX11504.9 : BOOL; (*STN 1 SLIDING DOOR - CLOSE (-160Y2) *)
	WY11501_10 AT  %MX11504.10 : BOOL; (*STN 1 SLIDING DOOR - CLOSE (-160Y2) *)
	WY11501_11 AT  %MX11504.11 : BOOL; (*STN 1 SLIDING DOOR - CLOSE (-160Y2) *)
	WY11501_12 AT  %MX11504.12 : BOOL; (*STN 1 SLIDING DOOR - CLOSE (-160Y2) *)
	WY11501_13 AT  %MX11504.13 : BOOL; (*STN 1 SLIDING DOOR - CLOSE (-160Y2) *)
	WY11501_14 AT  %MX11504.14 : BOOL; (*STN 1 SLIDING DOOR - CLOSE (-160Y2) *)
	WY11501_15 AT  %MX11504.15 : BOOL; (*STN 1 SLIDING DOOR - CLOSE (-160Y2) *)
	WY11501_16 AT  %MX11504.16 : BOOL; (*STN 1 SLIDING DOOR - CLOSE (-160Y2) *)
	WY11501_17 AT  %MX11504.17 : BOOL; (*STN 1 SLIDING DOOR - CLOSE (-160Y2) *)
	WY11501_18 AT  %MX11504.18 : BOOL; (*STN 1 SLIDING DOOR - CLOSE (-160Y2) *)
	WY11501_19 AT  %MX11504.19 : BOOL; (*STN 1 SLIDING DOOR - CLOSE (-160Y2) *)
	WY11501_20 AT  %MX11504.20 : BOOL; (*STN 1 SLIDING DOOR - CLOSE (-160Y2) *)
	WY11501_21 AT  %MX11504.21 : BOOL; (*STN 1 SLIDING DOOR - CLOSE (-160Y2) *)
	WY11501_22 AT  %MX11504.22 : BOOL; (*STN 1 SLIDING DOOR - CLOSE (-160Y2) *)
	WY11501_23 AT  %MX11504.23 : BOOL; (*STN 1 SLIDING DOOR - CLOSE (-160Y2) *)
	WY11501_24 AT  %MX11504.24 : BOOL; (*STN 1 SLIDING DOOR - CLOSE (-160Y2) *)
	WY11501_25 AT  %MX11504.25 : BOOL; (*STN 1 SLIDING DOOR - CLOSE (-160Y2) *)
	WY11501_26 AT  %MX11504.26 : BOOL; (*STN 1 SLIDING DOOR - CLOSE (-160Y2) *)
	WY11501_27 AT  %MX11504.27 : BOOL; (*STN 1 SLIDING DOOR - CLOSE (-160Y2) *)
	WY11501_28 AT  %MX11504.28 : BOOL; (*STN 1 SLIDING DOOR - CLOSE (-160Y2) *)
	WY11501_29 AT  %MX11504.29 : BOOL; (*STN 1 SLIDING DOOR - CLOSE (-160Y2) *)
	WY11501_30 AT  %MX11504.30 : BOOL; (*STN 1 SLIDING DOOR - CLOSE (-160Y2) *)
	WY11501_31 AT  %MX11504.31 : BOOL; (*STN 1 SLIDING DOOR - CLOSE (-160Y2) *)

	WY11502_00 AT  %MX11508.0 : BOOL; (*STN 4 SLIDING DOOR - OPEN (-160Y3) *)
	WY11502_01 AT  %MX11508.1 : BOOL; (*STN 4 SLIDING DOOR - OPEN (-160Y3) *)
	WY11502_02 AT  %MX11508.2 : BOOL; (*STN 4 SLIDING DOOR - OPEN (-160Y3) *)
	WY11502_03 AT  %MX11508.3 : BOOL; (*STN 4 SLIDING DOOR - OPEN (-160Y3) *)
	WY11502_04 AT  %MX11508.4 : BOOL; (*STN 4 SLIDING DOOR - OPEN (-160Y3) *)
	WY11502_05 AT  %MX11508.5 : BOOL; (*STN 4 SLIDING DOOR - OPEN (-160Y3) *)
	WY11502_06 AT  %MX11508.6 : BOOL; (*STN 4 SLIDING DOOR - OPEN (-160Y3) *)
	WY11502_07 AT  %MX11508.7 : BOOL; (*STN 4 SLIDING DOOR - OPEN (-160Y3) *)
	WY11502_08 AT  %MX11508.8 : BOOL; (*STN 4 SLIDING DOOR - OPEN (-160Y3) *)
	WY11502_09 AT  %MX11508.9 : BOOL; (*STN 4 SLIDING DOOR - OPEN (-160Y3) *)
	WY11502_10 AT  %MX11508.10 : BOOL; (*STN 4 SLIDING DOOR - OPEN (-160Y3) *)
	WY11502_11 AT  %MX11508.11 : BOOL; (*STN 4 SLIDING DOOR - OPEN (-160Y3) *)
	WY11502_12 AT  %MX11508.12 : BOOL; (*STN 4 SLIDING DOOR - OPEN (-160Y3) *)
	WY11502_13 AT  %MX11508.13 : BOOL; (*STN 4 SLIDING DOOR - OPEN (-160Y3) *)
	WY11502_14 AT  %MX11508.14 : BOOL; (*STN 4 SLIDING DOOR - OPEN (-160Y3) *)
	WY11502_15 AT  %MX11508.15 : BOOL; (*STN 4 SLIDING DOOR - OPEN (-160Y3) *)
	WY11502_16 AT  %MX11508.16 : BOOL; (*STN 4 SLIDING DOOR - OPEN (-160Y3) *)
	WY11502_17 AT  %MX11508.17 : BOOL; (*STN 4 SLIDING DOOR - OPEN (-160Y3) *)
	WY11502_18 AT  %MX11508.18 : BOOL; (*STN 4 SLIDING DOOR - OPEN (-160Y3) *)
	WY11502_19 AT  %MX11508.19 : BOOL; (*STN 4 SLIDING DOOR - OPEN (-160Y3) *)
	WY11502_20 AT  %MX11508.20 : BOOL; (*STN 4 SLIDING DOOR - OPEN (-160Y3) *)
	WY11502_21 AT  %MX11508.21 : BOOL; (*STN 4 SLIDING DOOR - OPEN (-160Y3) *)
	WY11502_22 AT  %MX11508.22 : BOOL; (*STN 4 SLIDING DOOR - OPEN (-160Y3) *)
	WY11502_23 AT  %MX11508.23 : BOOL; (*STN 4 SLIDING DOOR - OPEN (-160Y3) *)
	WY11502_24 AT  %MX11508.24 : BOOL; (*STN 4 SLIDING DOOR - OPEN (-160Y3) *)
	WY11502_25 AT  %MX11508.25 : BOOL; (*STN 4 SLIDING DOOR - OPEN (-160Y3) *)
	WY11502_26 AT  %MX11508.26 : BOOL; (*STN 4 SLIDING DOOR - OPEN (-160Y3) *)
	WY11502_27 AT  %MX11508.27 : BOOL; (*STN 4 SLIDING DOOR - OPEN (-160Y3) *)
	WY11502_28 AT  %MX11508.28 : BOOL; (*STN 4 SLIDING DOOR - OPEN (-160Y3) *)
	WY11502_29 AT  %MX11508.29 : BOOL; (*STN 4 SLIDING DOOR - OPEN (-160Y3) *)
	WY11502_30 AT  %MX11508.30 : BOOL; (*STN 4 SLIDING DOOR - OPEN (-160Y3) *)
	WY11502_31 AT  %MX11508.31 : BOOL; (*STN 4 SLIDING DOOR - OPEN (-160Y3) *)

	WY11503_00 AT  %MX11512.0 : BOOL; (*STN 4 SLIDING DOOR - CLOSE (-160Y4) *)
	WY11503_01 AT  %MX11512.1 : BOOL; (*STN 4 SLIDING DOOR - CLOSE (-160Y4) *)
	WY11503_02 AT  %MX11512.2 : BOOL; (*STN 4 SLIDING DOOR - CLOSE (-160Y4) *)
	WY11503_03 AT  %MX11512.3 : BOOL; (*STN 4 SLIDING DOOR - CLOSE (-160Y4) *)
	WY11503_04 AT  %MX11512.4 : BOOL; (*STN 4 SLIDING DOOR - CLOSE (-160Y4) *)
	WY11503_05 AT  %MX11512.5 : BOOL; (*STN 4 SLIDING DOOR - CLOSE (-160Y4) *)
	WY11503_06 AT  %MX11512.6 : BOOL; (*STN 4 SLIDING DOOR - CLOSE (-160Y4) *)
	WY11503_07 AT  %MX11512.7 : BOOL; (*STN 4 SLIDING DOOR - CLOSE (-160Y4) *)
	WY11503_08 AT  %MX11512.8 : BOOL; (*STN 4 SLIDING DOOR - CLOSE (-160Y4) *)
	WY11503_09 AT  %MX11512.9 : BOOL; (*STN 4 SLIDING DOOR - CLOSE (-160Y4) *)
	WY11503_10 AT  %MX11512.10 : BOOL; (*STN 4 SLIDING DOOR - CLOSE (-160Y4) *)
	WY11503_11 AT  %MX11512.11 : BOOL; (*STN 4 SLIDING DOOR - CLOSE (-160Y4) *)
	WY11503_12 AT  %MX11512.12 : BOOL; (*STN 4 SLIDING DOOR - CLOSE (-160Y4) *)
	WY11503_13 AT  %MX11512.13 : BOOL; (*STN 4 SLIDING DOOR - CLOSE (-160Y4) *)
	WY11503_14 AT  %MX11512.14 : BOOL; (*STN 4 SLIDING DOOR - CLOSE (-160Y4) *)
	WY11503_15 AT  %MX11512.15 : BOOL; (*STN 4 SLIDING DOOR - CLOSE (-160Y4) *)
	WY11503_16 AT  %MX11512.16 : BOOL; (*STN 4 SLIDING DOOR - CLOSE (-160Y4) *)
	WY11503_17 AT  %MX11512.17 : BOOL; (*STN 4 SLIDING DOOR - CLOSE (-160Y4) *)
	WY11503_18 AT  %MX11512.18 : BOOL; (*STN 4 SLIDING DOOR - CLOSE (-160Y4) *)
	WY11503_19 AT  %MX11512.19 : BOOL; (*STN 4 SLIDING DOOR - CLOSE (-160Y4) *)
	WY11503_20 AT  %MX11512.20 : BOOL; (*STN 4 SLIDING DOOR - CLOSE (-160Y4) *)
	WY11503_21 AT  %MX11512.21 : BOOL; (*STN 4 SLIDING DOOR - CLOSE (-160Y4) *)
	WY11503_22 AT  %MX11512.22 : BOOL; (*STN 4 SLIDING DOOR - CLOSE (-160Y4) *)
	WY11503_23 AT  %MX11512.23 : BOOL; (*STN 4 SLIDING DOOR - CLOSE (-160Y4) *)
	WY11503_24 AT  %MX11512.24 : BOOL; (*STN 4 SLIDING DOOR - CLOSE (-160Y4) *)
	WY11503_25 AT  %MX11512.25 : BOOL; (*STN 4 SLIDING DOOR - CLOSE (-160Y4) *)
	WY11503_26 AT  %MX11512.26 : BOOL; (*STN 4 SLIDING DOOR - CLOSE (-160Y4) *)
	WY11503_27 AT  %MX11512.27 : BOOL; (*STN 4 SLIDING DOOR - CLOSE (-160Y4) *)
	WY11503_28 AT  %MX11512.28 : BOOL; (*STN 4 SLIDING DOOR - CLOSE (-160Y4) *)
	WY11503_29 AT  %MX11512.29 : BOOL; (*STN 4 SLIDING DOOR - CLOSE (-160Y4) *)
	WY11503_30 AT  %MX11512.30 : BOOL; (*STN 4 SLIDING DOOR - CLOSE (-160Y4) *)
	WY11503_31 AT  %MX11512.31 : BOOL; (*STN 4 SLIDING DOOR - CLOSE (-160Y4) *)

	WY11504_00 AT  %MX11516.0 : BOOL; (*STN 5 SLIDING DOOR - OPEN (-160Y5) *)
	WY11504_01 AT  %MX11516.1 : BOOL; (*STN 5 SLIDING DOOR - OPEN (-160Y5) *)
	WY11504_02 AT  %MX11516.2 : BOOL; (*STN 5 SLIDING DOOR - OPEN (-160Y5) *)
	WY11504_03 AT  %MX11516.3 : BOOL; (*STN 5 SLIDING DOOR - OPEN (-160Y5) *)
	WY11504_04 AT  %MX11516.4 : BOOL; (*STN 5 SLIDING DOOR - OPEN (-160Y5) *)
	WY11504_05 AT  %MX11516.5 : BOOL; (*STN 5 SLIDING DOOR - OPEN (-160Y5) *)
	WY11504_06 AT  %MX11516.6 : BOOL; (*STN 5 SLIDING DOOR - OPEN (-160Y5) *)
	WY11504_07 AT  %MX11516.7 : BOOL; (*STN 5 SLIDING DOOR - OPEN (-160Y5) *)
	WY11504_08 AT  %MX11516.8 : BOOL; (*STN 5 SLIDING DOOR - OPEN (-160Y5) *)
	WY11504_09 AT  %MX11516.9 : BOOL; (*STN 5 SLIDING DOOR - OPEN (-160Y5) *)
	WY11504_10 AT  %MX11516.10 : BOOL; (*STN 5 SLIDING DOOR - OPEN (-160Y5) *)
	WY11504_11 AT  %MX11516.11 : BOOL; (*STN 5 SLIDING DOOR - OPEN (-160Y5) *)
	WY11504_12 AT  %MX11516.12 : BOOL; (*STN 5 SLIDING DOOR - OPEN (-160Y5) *)
	WY11504_13 AT  %MX11516.13 : BOOL; (*STN 5 SLIDING DOOR - OPEN (-160Y5) *)
	WY11504_14 AT  %MX11516.14 : BOOL; (*STN 5 SLIDING DOOR - OPEN (-160Y5) *)
	WY11504_15 AT  %MX11516.15 : BOOL; (*STN 5 SLIDING DOOR - OPEN (-160Y5) *)
	WY11504_16 AT  %MX11516.16 : BOOL; (*STN 5 SLIDING DOOR - OPEN (-160Y5) *)
	WY11504_17 AT  %MX11516.17 : BOOL; (*STN 5 SLIDING DOOR - OPEN (-160Y5) *)
	WY11504_18 AT  %MX11516.18 : BOOL; (*STN 5 SLIDING DOOR - OPEN (-160Y5) *)
	WY11504_19 AT  %MX11516.19 : BOOL; (*STN 5 SLIDING DOOR - OPEN (-160Y5) *)
	WY11504_20 AT  %MX11516.20 : BOOL; (*STN 5 SLIDING DOOR - OPEN (-160Y5) *)
	WY11504_21 AT  %MX11516.21 : BOOL; (*STN 5 SLIDING DOOR - OPEN (-160Y5) *)
	WY11504_22 AT  %MX11516.22 : BOOL; (*STN 5 SLIDING DOOR - OPEN (-160Y5) *)
	WY11504_23 AT  %MX11516.23 : BOOL; (*STN 5 SLIDING DOOR - OPEN (-160Y5) *)
	WY11504_24 AT  %MX11516.24 : BOOL; (*STN 5 SLIDING DOOR - OPEN (-160Y5) *)
	WY11504_25 AT  %MX11516.25 : BOOL; (*STN 5 SLIDING DOOR - OPEN (-160Y5) *)
	WY11504_26 AT  %MX11516.26 : BOOL; (*STN 5 SLIDING DOOR - OPEN (-160Y5) *)
	WY11504_27 AT  %MX11516.27 : BOOL; (*STN 5 SLIDING DOOR - OPEN (-160Y5) *)
	WY11504_28 AT  %MX11516.28 : BOOL; (*STN 5 SLIDING DOOR - OPEN (-160Y5) *)
	WY11504_29 AT  %MX11516.29 : BOOL; (*STN 5 SLIDING DOOR - OPEN (-160Y5) *)
	WY11504_30 AT  %MX11516.30 : BOOL; (*STN 5 SLIDING DOOR - OPEN (-160Y5) *)
	WY11504_31 AT  %MX11516.31 : BOOL; (*STN 5 SLIDING DOOR - OPEN (-160Y5) *)

	WY11505_00 AT  %MX11520.0 : BOOL; (*STN 5 SLIDING DOOR - CLOSE (-160Y6) *)
	WY11505_01 AT  %MX11520.1 : BOOL; (*STN 5 SLIDING DOOR - CLOSE (-160Y6) *)
	WY11505_02 AT  %MX11520.2 : BOOL; (*STN 5 SLIDING DOOR - CLOSE (-160Y6) *)
	WY11505_03 AT  %MX11520.3 : BOOL; (*STN 5 SLIDING DOOR - CLOSE (-160Y6) *)
	WY11505_04 AT  %MX11520.4 : BOOL; (*STN 5 SLIDING DOOR - CLOSE (-160Y6) *)
	WY11505_05 AT  %MX11520.5 : BOOL; (*STN 5 SLIDING DOOR - CLOSE (-160Y6) *)
	WY11505_06 AT  %MX11520.6 : BOOL; (*STN 5 SLIDING DOOR - CLOSE (-160Y6) *)
	WY11505_07 AT  %MX11520.7 : BOOL; (*STN 5 SLIDING DOOR - CLOSE (-160Y6) *)
	WY11505_08 AT  %MX11520.8 : BOOL; (*STN 5 SLIDING DOOR - CLOSE (-160Y6) *)
	WY11505_09 AT  %MX11520.9 : BOOL; (*STN 5 SLIDING DOOR - CLOSE (-160Y6) *)
	WY11505_10 AT  %MX11520.10 : BOOL; (*STN 5 SLIDING DOOR - CLOSE (-160Y6) *)
	WY11505_11 AT  %MX11520.11 : BOOL; (*STN 5 SLIDING DOOR - CLOSE (-160Y6) *)
	WY11505_12 AT  %MX11520.12 : BOOL; (*STN 5 SLIDING DOOR - CLOSE (-160Y6) *)
	WY11505_13 AT  %MX11520.13 : BOOL; (*STN 5 SLIDING DOOR - CLOSE (-160Y6) *)
	WY11505_14 AT  %MX11520.14 : BOOL; (*STN 5 SLIDING DOOR - CLOSE (-160Y6) *)
	WY11505_15 AT  %MX11520.15 : BOOL; (*STN 5 SLIDING DOOR - CLOSE (-160Y6) *)
	WY11505_16 AT  %MX11520.16 : BOOL; (*STN 5 SLIDING DOOR - CLOSE (-160Y6) *)
	WY11505_17 AT  %MX11520.17 : BOOL; (*STN 5 SLIDING DOOR - CLOSE (-160Y6) *)
	WY11505_18 AT  %MX11520.18 : BOOL; (*STN 5 SLIDING DOOR - CLOSE (-160Y6) *)
	WY11505_19 AT  %MX11520.19 : BOOL; (*STN 5 SLIDING DOOR - CLOSE (-160Y6) *)
	WY11505_20 AT  %MX11520.20 : BOOL; (*STN 5 SLIDING DOOR - CLOSE (-160Y6) *)
	WY11505_21 AT  %MX11520.21 : BOOL; (*STN 5 SLIDING DOOR - CLOSE (-160Y6) *)
	WY11505_22 AT  %MX11520.22 : BOOL; (*STN 5 SLIDING DOOR - CLOSE (-160Y6) *)
	WY11505_23 AT  %MX11520.23 : BOOL; (*STN 5 SLIDING DOOR - CLOSE (-160Y6) *)
	WY11505_24 AT  %MX11520.24 : BOOL; (*STN 5 SLIDING DOOR - CLOSE (-160Y6) *)
	WY11505_25 AT  %MX11520.25 : BOOL; (*STN 5 SLIDING DOOR - CLOSE (-160Y6) *)
	WY11505_26 AT  %MX11520.26 : BOOL; (*STN 5 SLIDING DOOR - CLOSE (-160Y6) *)
	WY11505_27 AT  %MX11520.27 : BOOL; (*STN 5 SLIDING DOOR - CLOSE (-160Y6) *)
	WY11505_28 AT  %MX11520.28 : BOOL; (*STN 5 SLIDING DOOR - CLOSE (-160Y6) *)
	WY11505_29 AT  %MX11520.29 : BOOL; (*STN 5 SLIDING DOOR - CLOSE (-160Y6) *)
	WY11505_30 AT  %MX11520.30 : BOOL; (*STN 5 SLIDING DOOR - CLOSE (-160Y6) *)
	WY11505_31 AT  %MX11520.31 : BOOL; (*STN 5 SLIDING DOOR - CLOSE (-160Y6) *)

	WY11506_00 AT  %MX11524.0 : BOOL; (*STN 5 SLIDING DOOR - CLAMP (-160Y7) *)
	WY11506_01 AT  %MX11524.1 : BOOL; (*STN 5 SLIDING DOOR - CLAMP (-160Y7) *)
	WY11506_02 AT  %MX11524.2 : BOOL; (*STN 5 SLIDING DOOR - CLAMP (-160Y7) *)
	WY11506_03 AT  %MX11524.3 : BOOL; (*STN 5 SLIDING DOOR - CLAMP (-160Y7) *)
	WY11506_04 AT  %MX11524.4 : BOOL; (*STN 5 SLIDING DOOR - CLAMP (-160Y7) *)
	WY11506_05 AT  %MX11524.5 : BOOL; (*STN 5 SLIDING DOOR - CLAMP (-160Y7) *)
	WY11506_06 AT  %MX11524.6 : BOOL; (*STN 5 SLIDING DOOR - CLAMP (-160Y7) *)
	WY11506_07 AT  %MX11524.7 : BOOL; (*STN 5 SLIDING DOOR - CLAMP (-160Y7) *)
	WY11506_08 AT  %MX11524.8 : BOOL; (*STN 5 SLIDING DOOR - CLAMP (-160Y7) *)
	WY11506_09 AT  %MX11524.9 : BOOL; (*STN 5 SLIDING DOOR - CLAMP (-160Y7) *)
	WY11506_10 AT  %MX11524.10 : BOOL; (*STN 5 SLIDING DOOR - CLAMP (-160Y7) *)
	WY11506_11 AT  %MX11524.11 : BOOL; (*STN 5 SLIDING DOOR - CLAMP (-160Y7) *)
	WY11506_12 AT  %MX11524.12 : BOOL; (*STN 5 SLIDING DOOR - CLAMP (-160Y7) *)
	WY11506_13 AT  %MX11524.13 : BOOL; (*STN 5 SLIDING DOOR - CLAMP (-160Y7) *)
	WY11506_14 AT  %MX11524.14 : BOOL; (*STN 5 SLIDING DOOR - CLAMP (-160Y7) *)
	WY11506_15 AT  %MX11524.15 : BOOL; (*STN 5 SLIDING DOOR - CLAMP (-160Y7) *)
	WY11506_16 AT  %MX11524.16 : BOOL; (*STN 5 SLIDING DOOR - CLAMP (-160Y7) *)
	WY11506_17 AT  %MX11524.17 : BOOL; (*STN 5 SLIDING DOOR - CLAMP (-160Y7) *)
	WY11506_18 AT  %MX11524.18 : BOOL; (*STN 5 SLIDING DOOR - CLAMP (-160Y7) *)
	WY11506_19 AT  %MX11524.19 : BOOL; (*STN 5 SLIDING DOOR - CLAMP (-160Y7) *)
	WY11506_20 AT  %MX11524.20 : BOOL; (*STN 5 SLIDING DOOR - CLAMP (-160Y7) *)
	WY11506_21 AT  %MX11524.21 : BOOL; (*STN 5 SLIDING DOOR - CLAMP (-160Y7) *)
	WY11506_22 AT  %MX11524.22 : BOOL; (*STN 5 SLIDING DOOR - CLAMP (-160Y7) *)
	WY11506_23 AT  %MX11524.23 : BOOL; (*STN 5 SLIDING DOOR - CLAMP (-160Y7) *)
	WY11506_24 AT  %MX11524.24 : BOOL; (*STN 5 SLIDING DOOR - CLAMP (-160Y7) *)
	WY11506_25 AT  %MX11524.25 : BOOL; (*STN 5 SLIDING DOOR - CLAMP (-160Y7) *)
	WY11506_26 AT  %MX11524.26 : BOOL; (*STN 5 SLIDING DOOR - CLAMP (-160Y7) *)
	WY11506_27 AT  %MX11524.27 : BOOL; (*STN 5 SLIDING DOOR - CLAMP (-160Y7) *)
	WY11506_28 AT  %MX11524.28 : BOOL; (*STN 5 SLIDING DOOR - CLAMP (-160Y7) *)
	WY11506_29 AT  %MX11524.29 : BOOL; (*STN 5 SLIDING DOOR - CLAMP (-160Y7) *)
	WY11506_30 AT  %MX11524.30 : BOOL; (*STN 5 SLIDING DOOR - CLAMP (-160Y7) *)
	WY11506_31 AT  %MX11524.31 : BOOL; (*STN 5 SLIDING DOOR - CLAMP (-160Y7) *)

	WY11507_00 AT  %MX11528.0 : BOOL; (*STN 5 SLIDING DOOR - UNCLAMP (-160Y8) *)
	WY11507_01 AT  %MX11528.1 : BOOL; (*STN 5 SLIDING DOOR - UNCLAMP (-160Y8) *)
	WY11507_02 AT  %MX11528.2 : BOOL; (*STN 5 SLIDING DOOR - UNCLAMP (-160Y8) *)
	WY11507_03 AT  %MX11528.3 : BOOL; (*STN 5 SLIDING DOOR - UNCLAMP (-160Y8) *)
	WY11507_04 AT  %MX11528.4 : BOOL; (*STN 5 SLIDING DOOR - UNCLAMP (-160Y8) *)
	WY11507_05 AT  %MX11528.5 : BOOL; (*STN 5 SLIDING DOOR - UNCLAMP (-160Y8) *)
	WY11507_06 AT  %MX11528.6 : BOOL; (*STN 5 SLIDING DOOR - UNCLAMP (-160Y8) *)
	WY11507_07 AT  %MX11528.7 : BOOL; (*STN 5 SLIDING DOOR - UNCLAMP (-160Y8) *)
	WY11507_08 AT  %MX11528.8 : BOOL; (*STN 5 SLIDING DOOR - UNCLAMP (-160Y8) *)
	WY11507_09 AT  %MX11528.9 : BOOL; (*STN 5 SLIDING DOOR - UNCLAMP (-160Y8) *)
	WY11507_10 AT  %MX11528.10 : BOOL; (*STN 5 SLIDING DOOR - UNCLAMP (-160Y8) *)
	WY11507_11 AT  %MX11528.11 : BOOL; (*STN 5 SLIDING DOOR - UNCLAMP (-160Y8) *)
	WY11507_12 AT  %MX11528.12 : BOOL; (*STN 5 SLIDING DOOR - UNCLAMP (-160Y8) *)
	WY11507_13 AT  %MX11528.13 : BOOL; (*STN 5 SLIDING DOOR - UNCLAMP (-160Y8) *)
	WY11507_14 AT  %MX11528.14 : BOOL; (*STN 5 SLIDING DOOR - UNCLAMP (-160Y8) *)
	WY11507_15 AT  %MX11528.15 : BOOL; (*STN 5 SLIDING DOOR - UNCLAMP (-160Y8) *)
	WY11507_16 AT  %MX11528.16 : BOOL; (*STN 5 SLIDING DOOR - UNCLAMP (-160Y8) *)
	WY11507_17 AT  %MX11528.17 : BOOL; (*STN 5 SLIDING DOOR - UNCLAMP (-160Y8) *)
	WY11507_18 AT  %MX11528.18 : BOOL; (*STN 5 SLIDING DOOR - UNCLAMP (-160Y8) *)
	WY11507_19 AT  %MX11528.19 : BOOL; (*STN 5 SLIDING DOOR - UNCLAMP (-160Y8) *)
	WY11507_20 AT  %MX11528.20 : BOOL; (*STN 5 SLIDING DOOR - UNCLAMP (-160Y8) *)
	WY11507_21 AT  %MX11528.21 : BOOL; (*STN 5 SLIDING DOOR - UNCLAMP (-160Y8) *)
	WY11507_22 AT  %MX11528.22 : BOOL; (*STN 5 SLIDING DOOR - UNCLAMP (-160Y8) *)
	WY11507_23 AT  %MX11528.23 : BOOL; (*STN 5 SLIDING DOOR - UNCLAMP (-160Y8) *)
	WY11507_24 AT  %MX11528.24 : BOOL; (*STN 5 SLIDING DOOR - UNCLAMP (-160Y8) *)
	WY11507_25 AT  %MX11528.25 : BOOL; (*STN 5 SLIDING DOOR - UNCLAMP (-160Y8) *)
	WY11507_26 AT  %MX11528.26 : BOOL; (*STN 5 SLIDING DOOR - UNCLAMP (-160Y8) *)
	WY11507_27 AT  %MX11528.27 : BOOL; (*STN 5 SLIDING DOOR - UNCLAMP (-160Y8) *)
	WY11507_28 AT  %MX11528.28 : BOOL; (*STN 5 SLIDING DOOR - UNCLAMP (-160Y8) *)
	WY11507_29 AT  %MX11528.29 : BOOL; (*STN 5 SLIDING DOOR - UNCLAMP (-160Y8) *)
	WY11507_30 AT  %MX11528.30 : BOOL; (*STN 5 SLIDING DOOR - UNCLAMP (-160Y8) *)
	WY11507_31 AT  %MX11528.31 : BOOL; (*STN 5 SLIDING DOOR - UNCLAMP (-160Y8) *)

	WY11508_00 AT  %MX11532.0 : BOOL; (*LD CYLINDER - UP (-160Y9) *)
	WY11508_01 AT  %MX11532.1 : BOOL; (*LD CYLINDER - UP (-160Y9) *)
	WY11508_02 AT  %MX11532.2 : BOOL; (*LD CYLINDER - UP (-160Y9) *)
	WY11508_03 AT  %MX11532.3 : BOOL; (*LD CYLINDER - UP (-160Y9) *)
	WY11508_04 AT  %MX11532.4 : BOOL; (*LD CYLINDER - UP (-160Y9) *)
	WY11508_05 AT  %MX11532.5 : BOOL; (*LD CYLINDER - UP (-160Y9) *)
	WY11508_06 AT  %MX11532.6 : BOOL; (*LD CYLINDER - UP (-160Y9) *)
	WY11508_07 AT  %MX11532.7 : BOOL; (*LD CYLINDER - UP (-160Y9) *)
	WY11508_08 AT  %MX11532.8 : BOOL; (*LD CYLINDER - UP (-160Y9) *)
	WY11508_09 AT  %MX11532.9 : BOOL; (*LD CYLINDER - UP (-160Y9) *)
	WY11508_10 AT  %MX11532.10 : BOOL; (*LD CYLINDER - UP (-160Y9) *)
	WY11508_11 AT  %MX11532.11 : BOOL; (*LD CYLINDER - UP (-160Y9) *)
	WY11508_12 AT  %MX11532.12 : BOOL; (*LD CYLINDER - UP (-160Y9) *)
	WY11508_13 AT  %MX11532.13 : BOOL; (*LD CYLINDER - UP (-160Y9) *)
	WY11508_14 AT  %MX11532.14 : BOOL; (*LD CYLINDER - UP (-160Y9) *)
	WY11508_15 AT  %MX11532.15 : BOOL; (*LD CYLINDER - UP (-160Y9) *)
	WY11508_16 AT  %MX11532.16 : BOOL; (*LD CYLINDER - UP (-160Y9) *)
	WY11508_17 AT  %MX11532.17 : BOOL; (*LD CYLINDER - UP (-160Y9) *)
	WY11508_18 AT  %MX11532.18 : BOOL; (*LD CYLINDER - UP (-160Y9) *)
	WY11508_19 AT  %MX11532.19 : BOOL; (*LD CYLINDER - UP (-160Y9) *)
	WY11508_20 AT  %MX11532.20 : BOOL; (*LD CYLINDER - UP (-160Y9) *)
	WY11508_21 AT  %MX11532.21 : BOOL; (*LD CYLINDER - UP (-160Y9) *)
	WY11508_22 AT  %MX11532.22 : BOOL; (*LD CYLINDER - UP (-160Y9) *)
	WY11508_23 AT  %MX11532.23 : BOOL; (*LD CYLINDER - UP (-160Y9) *)
	WY11508_24 AT  %MX11532.24 : BOOL; (*LD CYLINDER - UP (-160Y9) *)
	WY11508_25 AT  %MX11532.25 : BOOL; (*LD CYLINDER - UP (-160Y9) *)
	WY11508_26 AT  %MX11532.26 : BOOL; (*LD CYLINDER - UP (-160Y9) *)
	WY11508_27 AT  %MX11532.27 : BOOL; (*LD CYLINDER - UP (-160Y9) *)
	WY11508_28 AT  %MX11532.28 : BOOL; (*LD CYLINDER - UP (-160Y9) *)
	WY11508_29 AT  %MX11532.29 : BOOL; (*LD CYLINDER - UP (-160Y9) *)
	WY11508_30 AT  %MX11532.30 : BOOL; (*LD CYLINDER - UP (-160Y9) *)
	WY11508_31 AT  %MX11532.31 : BOOL; (*LD CYLINDER - UP (-160Y9) *)

	WY11509_00 AT  %MX11536.0 : BOOL; (*LD CYLINDER - DOWN (-160Y10) *)
	WY11509_01 AT  %MX11536.1 : BOOL; (*LD CYLINDER - DOWN (-160Y10) *)
	WY11509_02 AT  %MX11536.2 : BOOL; (*LD CYLINDER - DOWN (-160Y10) *)
	WY11509_03 AT  %MX11536.3 : BOOL; (*LD CYLINDER - DOWN (-160Y10) *)
	WY11509_04 AT  %MX11536.4 : BOOL; (*LD CYLINDER - DOWN (-160Y10) *)
	WY11509_05 AT  %MX11536.5 : BOOL; (*LD CYLINDER - DOWN (-160Y10) *)
	WY11509_06 AT  %MX11536.6 : BOOL; (*LD CYLINDER - DOWN (-160Y10) *)
	WY11509_07 AT  %MX11536.7 : BOOL; (*LD CYLINDER - DOWN (-160Y10) *)
	WY11509_08 AT  %MX11536.8 : BOOL; (*LD CYLINDER - DOWN (-160Y10) *)
	WY11509_09 AT  %MX11536.9 : BOOL; (*LD CYLINDER - DOWN (-160Y10) *)
	WY11509_10 AT  %MX11536.10 : BOOL; (*LD CYLINDER - DOWN (-160Y10) *)
	WY11509_11 AT  %MX11536.11 : BOOL; (*LD CYLINDER - DOWN (-160Y10) *)
	WY11509_12 AT  %MX11536.12 : BOOL; (*LD CYLINDER - DOWN (-160Y10) *)
	WY11509_13 AT  %MX11536.13 : BOOL; (*LD CYLINDER - DOWN (-160Y10) *)
	WY11509_14 AT  %MX11536.14 : BOOL; (*LD CYLINDER - DOWN (-160Y10) *)
	WY11509_15 AT  %MX11536.15 : BOOL; (*LD CYLINDER - DOWN (-160Y10) *)
	WY11509_16 AT  %MX11536.16 : BOOL; (*LD CYLINDER - DOWN (-160Y10) *)
	WY11509_17 AT  %MX11536.17 : BOOL; (*LD CYLINDER - DOWN (-160Y10) *)
	WY11509_18 AT  %MX11536.18 : BOOL; (*LD CYLINDER - DOWN (-160Y10) *)
	WY11509_19 AT  %MX11536.19 : BOOL; (*LD CYLINDER - DOWN (-160Y10) *)
	WY11509_20 AT  %MX11536.20 : BOOL; (*LD CYLINDER - DOWN (-160Y10) *)
	WY11509_21 AT  %MX11536.21 : BOOL; (*LD CYLINDER - DOWN (-160Y10) *)
	WY11509_22 AT  %MX11536.22 : BOOL; (*LD CYLINDER - DOWN (-160Y10) *)
	WY11509_23 AT  %MX11536.23 : BOOL; (*LD CYLINDER - DOWN (-160Y10) *)
	WY11509_24 AT  %MX11536.24 : BOOL; (*LD CYLINDER - DOWN (-160Y10) *)
	WY11509_25 AT  %MX11536.25 : BOOL; (*LD CYLINDER - DOWN (-160Y10) *)
	WY11509_26 AT  %MX11536.26 : BOOL; (*LD CYLINDER - DOWN (-160Y10) *)
	WY11509_27 AT  %MX11536.27 : BOOL; (*LD CYLINDER - DOWN (-160Y10) *)
	WY11509_28 AT  %MX11536.28 : BOOL; (*LD CYLINDER - DOWN (-160Y10) *)
	WY11509_29 AT  %MX11536.29 : BOOL; (*LD CYLINDER - DOWN (-160Y10) *)
	WY11509_30 AT  %MX11536.30 : BOOL; (*LD CYLINDER - DOWN (-160Y10) *)
	WY11509_31 AT  %MX11536.31 : BOOL; (*LD CYLINDER - DOWN (-160Y10) *)

	WY11510_00 AT  %MX11540.0 : BOOL; (*LD CYLINDER - FRONT (-160Y11) *)
	WY11510_01 AT  %MX11540.1 : BOOL; (*LD CYLINDER - FRONT (-160Y11) *)
	WY11510_02 AT  %MX11540.2 : BOOL; (*LD CYLINDER - FRONT (-160Y11) *)
	WY11510_03 AT  %MX11540.3 : BOOL; (*LD CYLINDER - FRONT (-160Y11) *)
	WY11510_04 AT  %MX11540.4 : BOOL; (*LD CYLINDER - FRONT (-160Y11) *)
	WY11510_05 AT  %MX11540.5 : BOOL; (*LD CYLINDER - FRONT (-160Y11) *)
	WY11510_06 AT  %MX11540.6 : BOOL; (*LD CYLINDER - FRONT (-160Y11) *)
	WY11510_07 AT  %MX11540.7 : BOOL; (*LD CYLINDER - FRONT (-160Y11) *)
	WY11510_08 AT  %MX11540.8 : BOOL; (*LD CYLINDER - FRONT (-160Y11) *)
	WY11510_09 AT  %MX11540.9 : BOOL; (*LD CYLINDER - FRONT (-160Y11) *)
	WY11510_10 AT  %MX11540.10 : BOOL; (*LD CYLINDER - FRONT (-160Y11) *)
	WY11510_11 AT  %MX11540.11 : BOOL; (*LD CYLINDER - FRONT (-160Y11) *)
	WY11510_12 AT  %MX11540.12 : BOOL; (*LD CYLINDER - FRONT (-160Y11) *)
	WY11510_13 AT  %MX11540.13 : BOOL; (*LD CYLINDER - FRONT (-160Y11) *)
	WY11510_14 AT  %MX11540.14 : BOOL; (*LD CYLINDER - FRONT (-160Y11) *)
	WY11510_15 AT  %MX11540.15 : BOOL; (*LD CYLINDER - FRONT (-160Y11) *)
	WY11510_16 AT  %MX11540.16 : BOOL; (*LD CYLINDER - FRONT (-160Y11) *)
	WY11510_17 AT  %MX11540.17 : BOOL; (*LD CYLINDER - FRONT (-160Y11) *)
	WY11510_18 AT  %MX11540.18 : BOOL; (*LD CYLINDER - FRONT (-160Y11) *)
	WY11510_19 AT  %MX11540.19 : BOOL; (*LD CYLINDER - FRONT (-160Y11) *)
	WY11510_20 AT  %MX11540.20 : BOOL; (*LD CYLINDER - FRONT (-160Y11) *)
	WY11510_21 AT  %MX11540.21 : BOOL; (*LD CYLINDER - FRONT (-160Y11) *)
	WY11510_22 AT  %MX11540.22 : BOOL; (*LD CYLINDER - FRONT (-160Y11) *)
	WY11510_23 AT  %MX11540.23 : BOOL; (*LD CYLINDER - FRONT (-160Y11) *)
	WY11510_24 AT  %MX11540.24 : BOOL; (*LD CYLINDER - FRONT (-160Y11) *)
	WY11510_25 AT  %MX11540.25 : BOOL; (*LD CYLINDER - FRONT (-160Y11) *)
	WY11510_26 AT  %MX11540.26 : BOOL; (*LD CYLINDER - FRONT (-160Y11) *)
	WY11510_27 AT  %MX11540.27 : BOOL; (*LD CYLINDER - FRONT (-160Y11) *)
	WY11510_28 AT  %MX11540.28 : BOOL; (*LD CYLINDER - FRONT (-160Y11) *)
	WY11510_29 AT  %MX11540.29 : BOOL; (*LD CYLINDER - FRONT (-160Y11) *)
	WY11510_30 AT  %MX11540.30 : BOOL; (*LD CYLINDER - FRONT (-160Y11) *)
	WY11510_31 AT  %MX11540.31 : BOOL; (*LD CYLINDER - FRONT (-160Y11) *)

	WY11511_00 AT  %MX11544.0 : BOOL; (*LD CYLINDER - BACK (-160Y12) *)
	WY11511_01 AT  %MX11544.1 : BOOL; (*LD CYLINDER - BACK (-160Y12) *)
	WY11511_02 AT  %MX11544.2 : BOOL; (*LD CYLINDER - BACK (-160Y12) *)
	WY11511_03 AT  %MX11544.3 : BOOL; (*LD CYLINDER - BACK (-160Y12) *)
	WY11511_04 AT  %MX11544.4 : BOOL; (*LD CYLINDER - BACK (-160Y12) *)
	WY11511_05 AT  %MX11544.5 : BOOL; (*LD CYLINDER - BACK (-160Y12) *)
	WY11511_06 AT  %MX11544.6 : BOOL; (*LD CYLINDER - BACK (-160Y12) *)
	WY11511_07 AT  %MX11544.7 : BOOL; (*LD CYLINDER - BACK (-160Y12) *)
	WY11511_08 AT  %MX11544.8 : BOOL; (*LD CYLINDER - BACK (-160Y12) *)
	WY11511_09 AT  %MX11544.9 : BOOL; (*LD CYLINDER - BACK (-160Y12) *)
	WY11511_10 AT  %MX11544.10 : BOOL; (*LD CYLINDER - BACK (-160Y12) *)
	WY11511_11 AT  %MX11544.11 : BOOL; (*LD CYLINDER - BACK (-160Y12) *)
	WY11511_12 AT  %MX11544.12 : BOOL; (*LD CYLINDER - BACK (-160Y12) *)
	WY11511_13 AT  %MX11544.13 : BOOL; (*LD CYLINDER - BACK (-160Y12) *)
	WY11511_14 AT  %MX11544.14 : BOOL; (*LD CYLINDER - BACK (-160Y12) *)
	WY11511_15 AT  %MX11544.15 : BOOL; (*LD CYLINDER - BACK (-160Y12) *)
	WY11511_16 AT  %MX11544.16 : BOOL; (*LD CYLINDER - BACK (-160Y12) *)
	WY11511_17 AT  %MX11544.17 : BOOL; (*LD CYLINDER - BACK (-160Y12) *)
	WY11511_18 AT  %MX11544.18 : BOOL; (*LD CYLINDER - BACK (-160Y12) *)
	WY11511_19 AT  %MX11544.19 : BOOL; (*LD CYLINDER - BACK (-160Y12) *)
	WY11511_20 AT  %MX11544.20 : BOOL; (*LD CYLINDER - BACK (-160Y12) *)
	WY11511_21 AT  %MX11544.21 : BOOL; (*LD CYLINDER - BACK (-160Y12) *)
	WY11511_22 AT  %MX11544.22 : BOOL; (*LD CYLINDER - BACK (-160Y12) *)
	WY11511_23 AT  %MX11544.23 : BOOL; (*LD CYLINDER - BACK (-160Y12) *)
	WY11511_24 AT  %MX11544.24 : BOOL; (*LD CYLINDER - BACK (-160Y12) *)
	WY11511_25 AT  %MX11544.25 : BOOL; (*LD CYLINDER - BACK (-160Y12) *)
	WY11511_26 AT  %MX11544.26 : BOOL; (*LD CYLINDER - BACK (-160Y12) *)
	WY11511_27 AT  %MX11544.27 : BOOL; (*LD CYLINDER - BACK (-160Y12) *)
	WY11511_28 AT  %MX11544.28 : BOOL; (*LD CYLINDER - BACK (-160Y12) *)
	WY11511_29 AT  %MX11544.29 : BOOL; (*LD CYLINDER - BACK (-160Y12) *)
	WY11511_30 AT  %MX11544.30 : BOOL; (*LD CYLINDER - BACK (-160Y12) *)
	WY11511_31 AT  %MX11544.31 : BOOL; (*LD CYLINDER - BACK (-160Y12) *)

	WY11512_00 AT  %MX11548.0 : BOOL; (*ULD CYLINDER - UP (-160Y13) *)
	WY11512_01 AT  %MX11548.1 : BOOL; (*ULD CYLINDER - UP (-160Y13) *)
	WY11512_02 AT  %MX11548.2 : BOOL; (*ULD CYLINDER - UP (-160Y13) *)
	WY11512_03 AT  %MX11548.3 : BOOL; (*ULD CYLINDER - UP (-160Y13) *)
	WY11512_04 AT  %MX11548.4 : BOOL; (*ULD CYLINDER - UP (-160Y13) *)
	WY11512_05 AT  %MX11548.5 : BOOL; (*ULD CYLINDER - UP (-160Y13) *)
	WY11512_06 AT  %MX11548.6 : BOOL; (*ULD CYLINDER - UP (-160Y13) *)
	WY11512_07 AT  %MX11548.7 : BOOL; (*ULD CYLINDER - UP (-160Y13) *)
	WY11512_08 AT  %MX11548.8 : BOOL; (*ULD CYLINDER - UP (-160Y13) *)
	WY11512_09 AT  %MX11548.9 : BOOL; (*ULD CYLINDER - UP (-160Y13) *)
	WY11512_10 AT  %MX11548.10 : BOOL; (*ULD CYLINDER - UP (-160Y13) *)
	WY11512_11 AT  %MX11548.11 : BOOL; (*ULD CYLINDER - UP (-160Y13) *)
	WY11512_12 AT  %MX11548.12 : BOOL; (*ULD CYLINDER - UP (-160Y13) *)
	WY11512_13 AT  %MX11548.13 : BOOL; (*ULD CYLINDER - UP (-160Y13) *)
	WY11512_14 AT  %MX11548.14 : BOOL; (*ULD CYLINDER - UP (-160Y13) *)
	WY11512_15 AT  %MX11548.15 : BOOL; (*ULD CYLINDER - UP (-160Y13) *)
	WY11512_16 AT  %MX11548.16 : BOOL; (*ULD CYLINDER - UP (-160Y13) *)
	WY11512_17 AT  %MX11548.17 : BOOL; (*ULD CYLINDER - UP (-160Y13) *)
	WY11512_18 AT  %MX11548.18 : BOOL; (*ULD CYLINDER - UP (-160Y13) *)
	WY11512_19 AT  %MX11548.19 : BOOL; (*ULD CYLINDER - UP (-160Y13) *)
	WY11512_20 AT  %MX11548.20 : BOOL; (*ULD CYLINDER - UP (-160Y13) *)
	WY11512_21 AT  %MX11548.21 : BOOL; (*ULD CYLINDER - UP (-160Y13) *)
	WY11512_22 AT  %MX11548.22 : BOOL; (*ULD CYLINDER - UP (-160Y13) *)
	WY11512_23 AT  %MX11548.23 : BOOL; (*ULD CYLINDER - UP (-160Y13) *)
	WY11512_24 AT  %MX11548.24 : BOOL; (*ULD CYLINDER - UP (-160Y13) *)
	WY11512_25 AT  %MX11548.25 : BOOL; (*ULD CYLINDER - UP (-160Y13) *)
	WY11512_26 AT  %MX11548.26 : BOOL; (*ULD CYLINDER - UP (-160Y13) *)
	WY11512_27 AT  %MX11548.27 : BOOL; (*ULD CYLINDER - UP (-160Y13) *)
	WY11512_28 AT  %MX11548.28 : BOOL; (*ULD CYLINDER - UP (-160Y13) *)
	WY11512_29 AT  %MX11548.29 : BOOL; (*ULD CYLINDER - UP (-160Y13) *)
	WY11512_30 AT  %MX11548.30 : BOOL; (*ULD CYLINDER - UP (-160Y13) *)
	WY11512_31 AT  %MX11548.31 : BOOL; (*ULD CYLINDER - UP (-160Y13) *)

	WY11513_00 AT  %MX11552.0 : BOOL; (*ULD CYLINDER - DOWN (-160Y14) *)
	WY11513_01 AT  %MX11552.1 : BOOL; (*ULD CYLINDER - DOWN (-160Y14) *)
	WY11513_02 AT  %MX11552.2 : BOOL; (*ULD CYLINDER - DOWN (-160Y14) *)
	WY11513_03 AT  %MX11552.3 : BOOL; (*ULD CYLINDER - DOWN (-160Y14) *)
	WY11513_04 AT  %MX11552.4 : BOOL; (*ULD CYLINDER - DOWN (-160Y14) *)
	WY11513_05 AT  %MX11552.5 : BOOL; (*ULD CYLINDER - DOWN (-160Y14) *)
	WY11513_06 AT  %MX11552.6 : BOOL; (*ULD CYLINDER - DOWN (-160Y14) *)
	WY11513_07 AT  %MX11552.7 : BOOL; (*ULD CYLINDER - DOWN (-160Y14) *)
	WY11513_08 AT  %MX11552.8 : BOOL; (*ULD CYLINDER - DOWN (-160Y14) *)
	WY11513_09 AT  %MX11552.9 : BOOL; (*ULD CYLINDER - DOWN (-160Y14) *)
	WY11513_10 AT  %MX11552.10 : BOOL; (*ULD CYLINDER - DOWN (-160Y14) *)
	WY11513_11 AT  %MX11552.11 : BOOL; (*ULD CYLINDER - DOWN (-160Y14) *)
	WY11513_12 AT  %MX11552.12 : BOOL; (*ULD CYLINDER - DOWN (-160Y14) *)
	WY11513_13 AT  %MX11552.13 : BOOL; (*ULD CYLINDER - DOWN (-160Y14) *)
	WY11513_14 AT  %MX11552.14 : BOOL; (*ULD CYLINDER - DOWN (-160Y14) *)
	WY11513_15 AT  %MX11552.15 : BOOL; (*ULD CYLINDER - DOWN (-160Y14) *)
	WY11513_16 AT  %MX11552.16 : BOOL; (*ULD CYLINDER - DOWN (-160Y14) *)
	WY11513_17 AT  %MX11552.17 : BOOL; (*ULD CYLINDER - DOWN (-160Y14) *)
	WY11513_18 AT  %MX11552.18 : BOOL; (*ULD CYLINDER - DOWN (-160Y14) *)
	WY11513_19 AT  %MX11552.19 : BOOL; (*ULD CYLINDER - DOWN (-160Y14) *)
	WY11513_20 AT  %MX11552.20 : BOOL; (*ULD CYLINDER - DOWN (-160Y14) *)
	WY11513_21 AT  %MX11552.21 : BOOL; (*ULD CYLINDER - DOWN (-160Y14) *)
	WY11513_22 AT  %MX11552.22 : BOOL; (*ULD CYLINDER - DOWN (-160Y14) *)
	WY11513_23 AT  %MX11552.23 : BOOL; (*ULD CYLINDER - DOWN (-160Y14) *)
	WY11513_24 AT  %MX11552.24 : BOOL; (*ULD CYLINDER - DOWN (-160Y14) *)
	WY11513_25 AT  %MX11552.25 : BOOL; (*ULD CYLINDER - DOWN (-160Y14) *)
	WY11513_26 AT  %MX11552.26 : BOOL; (*ULD CYLINDER - DOWN (-160Y14) *)
	WY11513_27 AT  %MX11552.27 : BOOL; (*ULD CYLINDER - DOWN (-160Y14) *)
	WY11513_28 AT  %MX11552.28 : BOOL; (*ULD CYLINDER - DOWN (-160Y14) *)
	WY11513_29 AT  %MX11552.29 : BOOL; (*ULD CYLINDER - DOWN (-160Y14) *)
	WY11513_30 AT  %MX11552.30 : BOOL; (*ULD CYLINDER - DOWN (-160Y14) *)
	WY11513_31 AT  %MX11552.31 : BOOL; (*ULD CYLINDER - DOWN (-160Y14) *)

	WY11514_00 AT  %MX11556.0 : BOOL; (*ULD CYLINDER - FRONT (-160Y15) *)
	WY11514_01 AT  %MX11556.1 : BOOL; (*ULD CYLINDER - FRONT (-160Y15) *)
	WY11514_02 AT  %MX11556.2 : BOOL; (*ULD CYLINDER - FRONT (-160Y15) *)
	WY11514_03 AT  %MX11556.3 : BOOL; (*ULD CYLINDER - FRONT (-160Y15) *)
	WY11514_04 AT  %MX11556.4 : BOOL; (*ULD CYLINDER - FRONT (-160Y15) *)
	WY11514_05 AT  %MX11556.5 : BOOL; (*ULD CYLINDER - FRONT (-160Y15) *)
	WY11514_06 AT  %MX11556.6 : BOOL; (*ULD CYLINDER - FRONT (-160Y15) *)
	WY11514_07 AT  %MX11556.7 : BOOL; (*ULD CYLINDER - FRONT (-160Y15) *)
	WY11514_08 AT  %MX11556.8 : BOOL; (*ULD CYLINDER - FRONT (-160Y15) *)
	WY11514_09 AT  %MX11556.9 : BOOL; (*ULD CYLINDER - FRONT (-160Y15) *)
	WY11514_10 AT  %MX11556.10 : BOOL; (*ULD CYLINDER - FRONT (-160Y15) *)
	WY11514_11 AT  %MX11556.11 : BOOL; (*ULD CYLINDER - FRONT (-160Y15) *)
	WY11514_12 AT  %MX11556.12 : BOOL; (*ULD CYLINDER - FRONT (-160Y15) *)
	WY11514_13 AT  %MX11556.13 : BOOL; (*ULD CYLINDER - FRONT (-160Y15) *)
	WY11514_14 AT  %MX11556.14 : BOOL; (*ULD CYLINDER - FRONT (-160Y15) *)
	WY11514_15 AT  %MX11556.15 : BOOL; (*ULD CYLINDER - FRONT (-160Y15) *)
	WY11514_16 AT  %MX11556.16 : BOOL; (*ULD CYLINDER - FRONT (-160Y15) *)
	WY11514_17 AT  %MX11556.17 : BOOL; (*ULD CYLINDER - FRONT (-160Y15) *)
	WY11514_18 AT  %MX11556.18 : BOOL; (*ULD CYLINDER - FRONT (-160Y15) *)
	WY11514_19 AT  %MX11556.19 : BOOL; (*ULD CYLINDER - FRONT (-160Y15) *)
	WY11514_20 AT  %MX11556.20 : BOOL; (*ULD CYLINDER - FRONT (-160Y15) *)
	WY11514_21 AT  %MX11556.21 : BOOL; (*ULD CYLINDER - FRONT (-160Y15) *)
	WY11514_22 AT  %MX11556.22 : BOOL; (*ULD CYLINDER - FRONT (-160Y15) *)
	WY11514_23 AT  %MX11556.23 : BOOL; (*ULD CYLINDER - FRONT (-160Y15) *)
	WY11514_24 AT  %MX11556.24 : BOOL; (*ULD CYLINDER - FRONT (-160Y15) *)
	WY11514_25 AT  %MX11556.25 : BOOL; (*ULD CYLINDER - FRONT (-160Y15) *)
	WY11514_26 AT  %MX11556.26 : BOOL; (*ULD CYLINDER - FRONT (-160Y15) *)
	WY11514_27 AT  %MX11556.27 : BOOL; (*ULD CYLINDER - FRONT (-160Y15) *)
	WY11514_28 AT  %MX11556.28 : BOOL; (*ULD CYLINDER - FRONT (-160Y15) *)
	WY11514_29 AT  %MX11556.29 : BOOL; (*ULD CYLINDER - FRONT (-160Y15) *)
	WY11514_30 AT  %MX11556.30 : BOOL; (*ULD CYLINDER - FRONT (-160Y15) *)
	WY11514_31 AT  %MX11556.31 : BOOL; (*ULD CYLINDER - FRONT (-160Y15) *)

	WY11515_00 AT  %MX11560.0 : BOOL; (*ULD CYLINDER - BACK (-160Y16) *)
	WY11515_01 AT  %MX11560.1 : BOOL; (*ULD CYLINDER - BACK (-160Y16) *)
	WY11515_02 AT  %MX11560.2 : BOOL; (*ULD CYLINDER - BACK (-160Y16) *)
	WY11515_03 AT  %MX11560.3 : BOOL; (*ULD CYLINDER - BACK (-160Y16) *)
	WY11515_04 AT  %MX11560.4 : BOOL; (*ULD CYLINDER - BACK (-160Y16) *)
	WY11515_05 AT  %MX11560.5 : BOOL; (*ULD CYLINDER - BACK (-160Y16) *)
	WY11515_06 AT  %MX11560.6 : BOOL; (*ULD CYLINDER - BACK (-160Y16) *)
	WY11515_07 AT  %MX11560.7 : BOOL; (*ULD CYLINDER - BACK (-160Y16) *)
	WY11515_08 AT  %MX11560.8 : BOOL; (*ULD CYLINDER - BACK (-160Y16) *)
	WY11515_09 AT  %MX11560.9 : BOOL; (*ULD CYLINDER - BACK (-160Y16) *)
	WY11515_10 AT  %MX11560.10 : BOOL; (*ULD CYLINDER - BACK (-160Y16) *)
	WY11515_11 AT  %MX11560.11 : BOOL; (*ULD CYLINDER - BACK (-160Y16) *)
	WY11515_12 AT  %MX11560.12 : BOOL; (*ULD CYLINDER - BACK (-160Y16) *)
	WY11515_13 AT  %MX11560.13 : BOOL; (*ULD CYLINDER - BACK (-160Y16) *)
	WY11515_14 AT  %MX11560.14 : BOOL; (*ULD CYLINDER - BACK (-160Y16) *)
	WY11515_15 AT  %MX11560.15 : BOOL; (*ULD CYLINDER - BACK (-160Y16) *)
	WY11515_16 AT  %MX11560.16 : BOOL; (*ULD CYLINDER - BACK (-160Y16) *)
	WY11515_17 AT  %MX11560.17 : BOOL; (*ULD CYLINDER - BACK (-160Y16) *)
	WY11515_18 AT  %MX11560.18 : BOOL; (*ULD CYLINDER - BACK (-160Y16) *)
	WY11515_19 AT  %MX11560.19 : BOOL; (*ULD CYLINDER - BACK (-160Y16) *)
	WY11515_20 AT  %MX11560.20 : BOOL; (*ULD CYLINDER - BACK (-160Y16) *)
	WY11515_21 AT  %MX11560.21 : BOOL; (*ULD CYLINDER - BACK (-160Y16) *)
	WY11515_22 AT  %MX11560.22 : BOOL; (*ULD CYLINDER - BACK (-160Y16) *)
	WY11515_23 AT  %MX11560.23 : BOOL; (*ULD CYLINDER - BACK (-160Y16) *)
	WY11515_24 AT  %MX11560.24 : BOOL; (*ULD CYLINDER - BACK (-160Y16) *)
	WY11515_25 AT  %MX11560.25 : BOOL; (*ULD CYLINDER - BACK (-160Y16) *)
	WY11515_26 AT  %MX11560.26 : BOOL; (*ULD CYLINDER - BACK (-160Y16) *)
	WY11515_27 AT  %MX11560.27 : BOOL; (*ULD CYLINDER - BACK (-160Y16) *)
	WY11515_28 AT  %MX11560.28 : BOOL; (*ULD CYLINDER - BACK (-160Y16) *)
	WY11515_29 AT  %MX11560.29 : BOOL; (*ULD CYLINDER - BACK (-160Y16) *)
	WY11515_30 AT  %MX11560.30 : BOOL; (*ULD CYLINDER - BACK (-160Y16) *)
	WY11515_31 AT  %MX11560.31 : BOOL; (*ULD CYLINDER - BACK (-160Y16) *)

	WY11600_00 AT  %MX11600.0 : BOOL; (*GENERAL INCOMING DIW SUPPLY AVINC-1 (-161Y1) *)
	WY11600_01 AT  %MX11600.1 : BOOL; (*GENERAL INCOMING DIW SUPPLY AVINC-1 (-161Y1) *)
	WY11600_02 AT  %MX11600.2 : BOOL; (*GENERAL INCOMING DIW SUPPLY AVINC-1 (-161Y1) *)
	WY11600_03 AT  %MX11600.3 : BOOL; (*GENERAL INCOMING DIW SUPPLY AVINC-1 (-161Y1) *)
	WY11600_04 AT  %MX11600.4 : BOOL; (*GENERAL INCOMING DIW SUPPLY AVINC-1 (-161Y1) *)
	WY11600_05 AT  %MX11600.5 : BOOL; (*GENERAL INCOMING DIW SUPPLY AVINC-1 (-161Y1) *)
	WY11600_06 AT  %MX11600.6 : BOOL; (*GENERAL INCOMING DIW SUPPLY AVINC-1 (-161Y1) *)
	WY11600_07 AT  %MX11600.7 : BOOL; (*GENERAL INCOMING DIW SUPPLY AVINC-1 (-161Y1) *)
	WY11600_08 AT  %MX11600.8 : BOOL; (*GENERAL INCOMING DIW SUPPLY AVINC-1 (-161Y1) *)
	WY11600_09 AT  %MX11600.9 : BOOL; (*GENERAL INCOMING DIW SUPPLY AVINC-1 (-161Y1) *)
	WY11600_10 AT  %MX11600.10 : BOOL; (*GENERAL INCOMING DIW SUPPLY AVINC-1 (-161Y1) *)
	WY11600_11 AT  %MX11600.11 : BOOL; (*GENERAL INCOMING DIW SUPPLY AVINC-1 (-161Y1) *)
	WY11600_12 AT  %MX11600.12 : BOOL; (*GENERAL INCOMING DIW SUPPLY AVINC-1 (-161Y1) *)
	WY11600_13 AT  %MX11600.13 : BOOL; (*GENERAL INCOMING DIW SUPPLY AVINC-1 (-161Y1) *)
	WY11600_14 AT  %MX11600.14 : BOOL; (*GENERAL INCOMING DIW SUPPLY AVINC-1 (-161Y1) *)
	WY11600_15 AT  %MX11600.15 : BOOL; (*GENERAL INCOMING DIW SUPPLY AVINC-1 (-161Y1) *)
	WY11600_16 AT  %MX11600.16 : BOOL; (*GENERAL INCOMING DIW SUPPLY AVINC-1 (-161Y1) *)
	WY11600_17 AT  %MX11600.17 : BOOL; (*GENERAL INCOMING DIW SUPPLY AVINC-1 (-161Y1) *)
	WY11600_18 AT  %MX11600.18 : BOOL; (*GENERAL INCOMING DIW SUPPLY AVINC-1 (-161Y1) *)
	WY11600_19 AT  %MX11600.19 : BOOL; (*GENERAL INCOMING DIW SUPPLY AVINC-1 (-161Y1) *)
	WY11600_20 AT  %MX11600.20 : BOOL; (*GENERAL INCOMING DIW SUPPLY AVINC-1 (-161Y1) *)
	WY11600_21 AT  %MX11600.21 : BOOL; (*GENERAL INCOMING DIW SUPPLY AVINC-1 (-161Y1) *)
	WY11600_22 AT  %MX11600.22 : BOOL; (*GENERAL INCOMING DIW SUPPLY AVINC-1 (-161Y1) *)
	WY11600_23 AT  %MX11600.23 : BOOL; (*GENERAL INCOMING DIW SUPPLY AVINC-1 (-161Y1) *)
	WY11600_24 AT  %MX11600.24 : BOOL; (*GENERAL INCOMING DIW SUPPLY AVINC-1 (-161Y1) *)
	WY11600_25 AT  %MX11600.25 : BOOL; (*GENERAL INCOMING DIW SUPPLY AVINC-1 (-161Y1) *)
	WY11600_26 AT  %MX11600.26 : BOOL; (*GENERAL INCOMING DIW SUPPLY AVINC-1 (-161Y1) *)
	WY11600_27 AT  %MX11600.27 : BOOL; (*GENERAL INCOMING DIW SUPPLY AVINC-1 (-161Y1) *)
	WY11600_28 AT  %MX11600.28 : BOOL; (*GENERAL INCOMING DIW SUPPLY AVINC-1 (-161Y1) *)
	WY11600_29 AT  %MX11600.29 : BOOL; (*GENERAL INCOMING DIW SUPPLY AVINC-1 (-161Y1) *)
	WY11600_30 AT  %MX11600.30 : BOOL; (*GENERAL INCOMING DIW SUPPLY AVINC-1 (-161Y1) *)
	WY11600_31 AT  %MX11600.31 : BOOL; (*GENERAL INCOMING DIW SUPPLY AVINC-1 (-161Y1) *)

	WY11601_00 AT  %MX11604.0 : BOOL; (*STN 1 PROCESS TANK INCOMING DI SUPPLY AV1-1 (-161Y2) *)
	WY11601_01 AT  %MX11604.1 : BOOL; (*STN 1 PROCESS TANK INCOMING DI SUPPLY AV1-1 (-161Y2) *)
	WY11601_02 AT  %MX11604.2 : BOOL; (*STN 1 PROCESS TANK INCOMING DI SUPPLY AV1-1 (-161Y2) *)
	WY11601_03 AT  %MX11604.3 : BOOL; (*STN 1 PROCESS TANK INCOMING DI SUPPLY AV1-1 (-161Y2) *)
	WY11601_04 AT  %MX11604.4 : BOOL; (*STN 1 PROCESS TANK INCOMING DI SUPPLY AV1-1 (-161Y2) *)
	WY11601_05 AT  %MX11604.5 : BOOL; (*STN 1 PROCESS TANK INCOMING DI SUPPLY AV1-1 (-161Y2) *)
	WY11601_06 AT  %MX11604.6 : BOOL; (*STN 1 PROCESS TANK INCOMING DI SUPPLY AV1-1 (-161Y2) *)
	WY11601_07 AT  %MX11604.7 : BOOL; (*STN 1 PROCESS TANK INCOMING DI SUPPLY AV1-1 (-161Y2) *)
	WY11601_08 AT  %MX11604.8 : BOOL; (*STN 1 PROCESS TANK INCOMING DI SUPPLY AV1-1 (-161Y2) *)
	WY11601_09 AT  %MX11604.9 : BOOL; (*STN 1 PROCESS TANK INCOMING DI SUPPLY AV1-1 (-161Y2) *)
	WY11601_10 AT  %MX11604.10 : BOOL; (*STN 1 PROCESS TANK INCOMING DI SUPPLY AV1-1 (-161Y2) *)
	WY11601_11 AT  %MX11604.11 : BOOL; (*STN 1 PROCESS TANK INCOMING DI SUPPLY AV1-1 (-161Y2) *)
	WY11601_12 AT  %MX11604.12 : BOOL; (*STN 1 PROCESS TANK INCOMING DI SUPPLY AV1-1 (-161Y2) *)
	WY11601_13 AT  %MX11604.13 : BOOL; (*STN 1 PROCESS TANK INCOMING DI SUPPLY AV1-1 (-161Y2) *)
	WY11601_14 AT  %MX11604.14 : BOOL; (*STN 1 PROCESS TANK INCOMING DI SUPPLY AV1-1 (-161Y2) *)
	WY11601_15 AT  %MX11604.15 : BOOL; (*STN 1 PROCESS TANK INCOMING DI SUPPLY AV1-1 (-161Y2) *)
	WY11601_16 AT  %MX11604.16 : BOOL; (*STN 1 PROCESS TANK INCOMING DI SUPPLY AV1-1 (-161Y2) *)
	WY11601_17 AT  %MX11604.17 : BOOL; (*STN 1 PROCESS TANK INCOMING DI SUPPLY AV1-1 (-161Y2) *)
	WY11601_18 AT  %MX11604.18 : BOOL; (*STN 1 PROCESS TANK INCOMING DI SUPPLY AV1-1 (-161Y2) *)
	WY11601_19 AT  %MX11604.19 : BOOL; (*STN 1 PROCESS TANK INCOMING DI SUPPLY AV1-1 (-161Y2) *)
	WY11601_20 AT  %MX11604.20 : BOOL; (*STN 1 PROCESS TANK INCOMING DI SUPPLY AV1-1 (-161Y2) *)
	WY11601_21 AT  %MX11604.21 : BOOL; (*STN 1 PROCESS TANK INCOMING DI SUPPLY AV1-1 (-161Y2) *)
	WY11601_22 AT  %MX11604.22 : BOOL; (*STN 1 PROCESS TANK INCOMING DI SUPPLY AV1-1 (-161Y2) *)
	WY11601_23 AT  %MX11604.23 : BOOL; (*STN 1 PROCESS TANK INCOMING DI SUPPLY AV1-1 (-161Y2) *)
	WY11601_24 AT  %MX11604.24 : BOOL; (*STN 1 PROCESS TANK INCOMING DI SUPPLY AV1-1 (-161Y2) *)
	WY11601_25 AT  %MX11604.25 : BOOL; (*STN 1 PROCESS TANK INCOMING DI SUPPLY AV1-1 (-161Y2) *)
	WY11601_26 AT  %MX11604.26 : BOOL; (*STN 1 PROCESS TANK INCOMING DI SUPPLY AV1-1 (-161Y2) *)
	WY11601_27 AT  %MX11604.27 : BOOL; (*STN 1 PROCESS TANK INCOMING DI SUPPLY AV1-1 (-161Y2) *)
	WY11601_28 AT  %MX11604.28 : BOOL; (*STN 1 PROCESS TANK INCOMING DI SUPPLY AV1-1 (-161Y2) *)
	WY11601_29 AT  %MX11604.29 : BOOL; (*STN 1 PROCESS TANK INCOMING DI SUPPLY AV1-1 (-161Y2) *)
	WY11601_30 AT  %MX11604.30 : BOOL; (*STN 1 PROCESS TANK INCOMING DI SUPPLY AV1-1 (-161Y2) *)
	WY11601_31 AT  %MX11604.31 : BOOL; (*STN 1 PROCESS TANK INCOMING DI SUPPLY AV1-1 (-161Y2) *)

	WY11602_00 AT  %MX11608.0 : BOOL; (*STN 1 SUB TANK INCOMING DIW SUPPLY AV1-2 (-161Y3) *)
	WY11602_01 AT  %MX11608.1 : BOOL; (*STN 1 SUB TANK INCOMING DIW SUPPLY AV1-2 (-161Y3) *)
	WY11602_02 AT  %MX11608.2 : BOOL; (*STN 1 SUB TANK INCOMING DIW SUPPLY AV1-2 (-161Y3) *)
	WY11602_03 AT  %MX11608.3 : BOOL; (*STN 1 SUB TANK INCOMING DIW SUPPLY AV1-2 (-161Y3) *)
	WY11602_04 AT  %MX11608.4 : BOOL; (*STN 1 SUB TANK INCOMING DIW SUPPLY AV1-2 (-161Y3) *)
	WY11602_05 AT  %MX11608.5 : BOOL; (*STN 1 SUB TANK INCOMING DIW SUPPLY AV1-2 (-161Y3) *)
	WY11602_06 AT  %MX11608.6 : BOOL; (*STN 1 SUB TANK INCOMING DIW SUPPLY AV1-2 (-161Y3) *)
	WY11602_07 AT  %MX11608.7 : BOOL; (*STN 1 SUB TANK INCOMING DIW SUPPLY AV1-2 (-161Y3) *)
	WY11602_08 AT  %MX11608.8 : BOOL; (*STN 1 SUB TANK INCOMING DIW SUPPLY AV1-2 (-161Y3) *)
	WY11602_09 AT  %MX11608.9 : BOOL; (*STN 1 SUB TANK INCOMING DIW SUPPLY AV1-2 (-161Y3) *)
	WY11602_10 AT  %MX11608.10 : BOOL; (*STN 1 SUB TANK INCOMING DIW SUPPLY AV1-2 (-161Y3) *)
	WY11602_11 AT  %MX11608.11 : BOOL; (*STN 1 SUB TANK INCOMING DIW SUPPLY AV1-2 (-161Y3) *)
	WY11602_12 AT  %MX11608.12 : BOOL; (*STN 1 SUB TANK INCOMING DIW SUPPLY AV1-2 (-161Y3) *)
	WY11602_13 AT  %MX11608.13 : BOOL; (*STN 1 SUB TANK INCOMING DIW SUPPLY AV1-2 (-161Y3) *)
	WY11602_14 AT  %MX11608.14 : BOOL; (*STN 1 SUB TANK INCOMING DIW SUPPLY AV1-2 (-161Y3) *)
	WY11602_15 AT  %MX11608.15 : BOOL; (*STN 1 SUB TANK INCOMING DIW SUPPLY AV1-2 (-161Y3) *)
	WY11602_16 AT  %MX11608.16 : BOOL; (*STN 1 SUB TANK INCOMING DIW SUPPLY AV1-2 (-161Y3) *)
	WY11602_17 AT  %MX11608.17 : BOOL; (*STN 1 SUB TANK INCOMING DIW SUPPLY AV1-2 (-161Y3) *)
	WY11602_18 AT  %MX11608.18 : BOOL; (*STN 1 SUB TANK INCOMING DIW SUPPLY AV1-2 (-161Y3) *)
	WY11602_19 AT  %MX11608.19 : BOOL; (*STN 1 SUB TANK INCOMING DIW SUPPLY AV1-2 (-161Y3) *)
	WY11602_20 AT  %MX11608.20 : BOOL; (*STN 1 SUB TANK INCOMING DIW SUPPLY AV1-2 (-161Y3) *)
	WY11602_21 AT  %MX11608.21 : BOOL; (*STN 1 SUB TANK INCOMING DIW SUPPLY AV1-2 (-161Y3) *)
	WY11602_22 AT  %MX11608.22 : BOOL; (*STN 1 SUB TANK INCOMING DIW SUPPLY AV1-2 (-161Y3) *)
	WY11602_23 AT  %MX11608.23 : BOOL; (*STN 1 SUB TANK INCOMING DIW SUPPLY AV1-2 (-161Y3) *)
	WY11602_24 AT  %MX11608.24 : BOOL; (*STN 1 SUB TANK INCOMING DIW SUPPLY AV1-2 (-161Y3) *)
	WY11602_25 AT  %MX11608.25 : BOOL; (*STN 1 SUB TANK INCOMING DIW SUPPLY AV1-2 (-161Y3) *)
	WY11602_26 AT  %MX11608.26 : BOOL; (*STN 1 SUB TANK INCOMING DIW SUPPLY AV1-2 (-161Y3) *)
	WY11602_27 AT  %MX11608.27 : BOOL; (*STN 1 SUB TANK INCOMING DIW SUPPLY AV1-2 (-161Y3) *)
	WY11602_28 AT  %MX11608.28 : BOOL; (*STN 1 SUB TANK INCOMING DIW SUPPLY AV1-2 (-161Y3) *)
	WY11602_29 AT  %MX11608.29 : BOOL; (*STN 1 SUB TANK INCOMING DIW SUPPLY AV1-2 (-161Y3) *)
	WY11602_30 AT  %MX11608.30 : BOOL; (*STN 1 SUB TANK INCOMING DIW SUPPLY AV1-2 (-161Y3) *)
	WY11602_31 AT  %MX11608.31 : BOOL; (*STN 1 SUB TANK INCOMING DIW SUPPLY AV1-2 (-161Y3) *)

	WY11603_00 AT  %MX11612.0 : BOOL; (*STN 1 DETERGENT SUPPLY 3-2 WAY AV1-3 (-161Y4) *)
	WY11603_01 AT  %MX11612.1 : BOOL; (*STN 1 DETERGENT SUPPLY 3-2 WAY AV1-3 (-161Y4) *)
	WY11603_02 AT  %MX11612.2 : BOOL; (*STN 1 DETERGENT SUPPLY 3-2 WAY AV1-3 (-161Y4) *)
	WY11603_03 AT  %MX11612.3 : BOOL; (*STN 1 DETERGENT SUPPLY 3-2 WAY AV1-3 (-161Y4) *)
	WY11603_04 AT  %MX11612.4 : BOOL; (*STN 1 DETERGENT SUPPLY 3-2 WAY AV1-3 (-161Y4) *)
	WY11603_05 AT  %MX11612.5 : BOOL; (*STN 1 DETERGENT SUPPLY 3-2 WAY AV1-3 (-161Y4) *)
	WY11603_06 AT  %MX11612.6 : BOOL; (*STN 1 DETERGENT SUPPLY 3-2 WAY AV1-3 (-161Y4) *)
	WY11603_07 AT  %MX11612.7 : BOOL; (*STN 1 DETERGENT SUPPLY 3-2 WAY AV1-3 (-161Y4) *)
	WY11603_08 AT  %MX11612.8 : BOOL; (*STN 1 DETERGENT SUPPLY 3-2 WAY AV1-3 (-161Y4) *)
	WY11603_09 AT  %MX11612.9 : BOOL; (*STN 1 DETERGENT SUPPLY 3-2 WAY AV1-3 (-161Y4) *)
	WY11603_10 AT  %MX11612.10 : BOOL; (*STN 1 DETERGENT SUPPLY 3-2 WAY AV1-3 (-161Y4) *)
	WY11603_11 AT  %MX11612.11 : BOOL; (*STN 1 DETERGENT SUPPLY 3-2 WAY AV1-3 (-161Y4) *)
	WY11603_12 AT  %MX11612.12 : BOOL; (*STN 1 DETERGENT SUPPLY 3-2 WAY AV1-3 (-161Y4) *)
	WY11603_13 AT  %MX11612.13 : BOOL; (*STN 1 DETERGENT SUPPLY 3-2 WAY AV1-3 (-161Y4) *)
	WY11603_14 AT  %MX11612.14 : BOOL; (*STN 1 DETERGENT SUPPLY 3-2 WAY AV1-3 (-161Y4) *)
	WY11603_15 AT  %MX11612.15 : BOOL; (*STN 1 DETERGENT SUPPLY 3-2 WAY AV1-3 (-161Y4) *)
	WY11603_16 AT  %MX11612.16 : BOOL; (*STN 1 DETERGENT SUPPLY 3-2 WAY AV1-3 (-161Y4) *)
	WY11603_17 AT  %MX11612.17 : BOOL; (*STN 1 DETERGENT SUPPLY 3-2 WAY AV1-3 (-161Y4) *)
	WY11603_18 AT  %MX11612.18 : BOOL; (*STN 1 DETERGENT SUPPLY 3-2 WAY AV1-3 (-161Y4) *)
	WY11603_19 AT  %MX11612.19 : BOOL; (*STN 1 DETERGENT SUPPLY 3-2 WAY AV1-3 (-161Y4) *)
	WY11603_20 AT  %MX11612.20 : BOOL; (*STN 1 DETERGENT SUPPLY 3-2 WAY AV1-3 (-161Y4) *)
	WY11603_21 AT  %MX11612.21 : BOOL; (*STN 1 DETERGENT SUPPLY 3-2 WAY AV1-3 (-161Y4) *)
	WY11603_22 AT  %MX11612.22 : BOOL; (*STN 1 DETERGENT SUPPLY 3-2 WAY AV1-3 (-161Y4) *)
	WY11603_23 AT  %MX11612.23 : BOOL; (*STN 1 DETERGENT SUPPLY 3-2 WAY AV1-3 (-161Y4) *)
	WY11603_24 AT  %MX11612.24 : BOOL; (*STN 1 DETERGENT SUPPLY 3-2 WAY AV1-3 (-161Y4) *)
	WY11603_25 AT  %MX11612.25 : BOOL; (*STN 1 DETERGENT SUPPLY 3-2 WAY AV1-3 (-161Y4) *)
	WY11603_26 AT  %MX11612.26 : BOOL; (*STN 1 DETERGENT SUPPLY 3-2 WAY AV1-3 (-161Y4) *)
	WY11603_27 AT  %MX11612.27 : BOOL; (*STN 1 DETERGENT SUPPLY 3-2 WAY AV1-3 (-161Y4) *)
	WY11603_28 AT  %MX11612.28 : BOOL; (*STN 1 DETERGENT SUPPLY 3-2 WAY AV1-3 (-161Y4) *)
	WY11603_29 AT  %MX11612.29 : BOOL; (*STN 1 DETERGENT SUPPLY 3-2 WAY AV1-3 (-161Y4) *)
	WY11603_30 AT  %MX11612.30 : BOOL; (*STN 1 DETERGENT SUPPLY 3-2 WAY AV1-3 (-161Y4) *)
	WY11603_31 AT  %MX11612.31 : BOOL; (*STN 1 DETERGENT SUPPLY 3-2 WAY AV1-3 (-161Y4) *)

	WY11604_00 AT  %MX11616.0 : BOOL; (*STN 2 PROCESS TANK INCOMING DIW SUPPLY AV2-1 (-161Y5) *)
	WY11604_01 AT  %MX11616.1 : BOOL; (*STN 2 PROCESS TANK INCOMING DIW SUPPLY AV2-1 (-161Y5) *)
	WY11604_02 AT  %MX11616.2 : BOOL; (*STN 2 PROCESS TANK INCOMING DIW SUPPLY AV2-1 (-161Y5) *)
	WY11604_03 AT  %MX11616.3 : BOOL; (*STN 2 PROCESS TANK INCOMING DIW SUPPLY AV2-1 (-161Y5) *)
	WY11604_04 AT  %MX11616.4 : BOOL; (*STN 2 PROCESS TANK INCOMING DIW SUPPLY AV2-1 (-161Y5) *)
	WY11604_05 AT  %MX11616.5 : BOOL; (*STN 2 PROCESS TANK INCOMING DIW SUPPLY AV2-1 (-161Y5) *)
	WY11604_06 AT  %MX11616.6 : BOOL; (*STN 2 PROCESS TANK INCOMING DIW SUPPLY AV2-1 (-161Y5) *)
	WY11604_07 AT  %MX11616.7 : BOOL; (*STN 2 PROCESS TANK INCOMING DIW SUPPLY AV2-1 (-161Y5) *)
	WY11604_08 AT  %MX11616.8 : BOOL; (*STN 2 PROCESS TANK INCOMING DIW SUPPLY AV2-1 (-161Y5) *)
	WY11604_09 AT  %MX11616.9 : BOOL; (*STN 2 PROCESS TANK INCOMING DIW SUPPLY AV2-1 (-161Y5) *)
	WY11604_10 AT  %MX11616.10 : BOOL; (*STN 2 PROCESS TANK INCOMING DIW SUPPLY AV2-1 (-161Y5) *)
	WY11604_11 AT  %MX11616.11 : BOOL; (*STN 2 PROCESS TANK INCOMING DIW SUPPLY AV2-1 (-161Y5) *)
	WY11604_12 AT  %MX11616.12 : BOOL; (*STN 2 PROCESS TANK INCOMING DIW SUPPLY AV2-1 (-161Y5) *)
	WY11604_13 AT  %MX11616.13 : BOOL; (*STN 2 PROCESS TANK INCOMING DIW SUPPLY AV2-1 (-161Y5) *)
	WY11604_14 AT  %MX11616.14 : BOOL; (*STN 2 PROCESS TANK INCOMING DIW SUPPLY AV2-1 (-161Y5) *)
	WY11604_15 AT  %MX11616.15 : BOOL; (*STN 2 PROCESS TANK INCOMING DIW SUPPLY AV2-1 (-161Y5) *)
	WY11604_16 AT  %MX11616.16 : BOOL; (*STN 2 PROCESS TANK INCOMING DIW SUPPLY AV2-1 (-161Y5) *)
	WY11604_17 AT  %MX11616.17 : BOOL; (*STN 2 PROCESS TANK INCOMING DIW SUPPLY AV2-1 (-161Y5) *)
	WY11604_18 AT  %MX11616.18 : BOOL; (*STN 2 PROCESS TANK INCOMING DIW SUPPLY AV2-1 (-161Y5) *)
	WY11604_19 AT  %MX11616.19 : BOOL; (*STN 2 PROCESS TANK INCOMING DIW SUPPLY AV2-1 (-161Y5) *)
	WY11604_20 AT  %MX11616.20 : BOOL; (*STN 2 PROCESS TANK INCOMING DIW SUPPLY AV2-1 (-161Y5) *)
	WY11604_21 AT  %MX11616.21 : BOOL; (*STN 2 PROCESS TANK INCOMING DIW SUPPLY AV2-1 (-161Y5) *)
	WY11604_22 AT  %MX11616.22 : BOOL; (*STN 2 PROCESS TANK INCOMING DIW SUPPLY AV2-1 (-161Y5) *)
	WY11604_23 AT  %MX11616.23 : BOOL; (*STN 2 PROCESS TANK INCOMING DIW SUPPLY AV2-1 (-161Y5) *)
	WY11604_24 AT  %MX11616.24 : BOOL; (*STN 2 PROCESS TANK INCOMING DIW SUPPLY AV2-1 (-161Y5) *)
	WY11604_25 AT  %MX11616.25 : BOOL; (*STN 2 PROCESS TANK INCOMING DIW SUPPLY AV2-1 (-161Y5) *)
	WY11604_26 AT  %MX11616.26 : BOOL; (*STN 2 PROCESS TANK INCOMING DIW SUPPLY AV2-1 (-161Y5) *)
	WY11604_27 AT  %MX11616.27 : BOOL; (*STN 2 PROCESS TANK INCOMING DIW SUPPLY AV2-1 (-161Y5) *)
	WY11604_28 AT  %MX11616.28 : BOOL; (*STN 2 PROCESS TANK INCOMING DIW SUPPLY AV2-1 (-161Y5) *)
	WY11604_29 AT  %MX11616.29 : BOOL; (*STN 2 PROCESS TANK INCOMING DIW SUPPLY AV2-1 (-161Y5) *)
	WY11604_30 AT  %MX11616.30 : BOOL; (*STN 2 PROCESS TANK INCOMING DIW SUPPLY AV2-1 (-161Y5) *)
	WY11604_31 AT  %MX11616.31 : BOOL; (*STN 2 PROCESS TANK INCOMING DIW SUPPLY AV2-1 (-161Y5) *)

	WY11605_00 AT  %MX11620.0 : BOOL; (*STN 3 PROCESS TANK INCOMING DIW SUPPLY AV3-1 (-161Y6) *)
	WY11605_01 AT  %MX11620.1 : BOOL; (*STN 3 PROCESS TANK INCOMING DIW SUPPLY AV3-1 (-161Y6) *)
	WY11605_02 AT  %MX11620.2 : BOOL; (*STN 3 PROCESS TANK INCOMING DIW SUPPLY AV3-1 (-161Y6) *)
	WY11605_03 AT  %MX11620.3 : BOOL; (*STN 3 PROCESS TANK INCOMING DIW SUPPLY AV3-1 (-161Y6) *)
	WY11605_04 AT  %MX11620.4 : BOOL; (*STN 3 PROCESS TANK INCOMING DIW SUPPLY AV3-1 (-161Y6) *)
	WY11605_05 AT  %MX11620.5 : BOOL; (*STN 3 PROCESS TANK INCOMING DIW SUPPLY AV3-1 (-161Y6) *)
	WY11605_06 AT  %MX11620.6 : BOOL; (*STN 3 PROCESS TANK INCOMING DIW SUPPLY AV3-1 (-161Y6) *)
	WY11605_07 AT  %MX11620.7 : BOOL; (*STN 3 PROCESS TANK INCOMING DIW SUPPLY AV3-1 (-161Y6) *)
	WY11605_08 AT  %MX11620.8 : BOOL; (*STN 3 PROCESS TANK INCOMING DIW SUPPLY AV3-1 (-161Y6) *)
	WY11605_09 AT  %MX11620.9 : BOOL; (*STN 3 PROCESS TANK INCOMING DIW SUPPLY AV3-1 (-161Y6) *)
	WY11605_10 AT  %MX11620.10 : BOOL; (*STN 3 PROCESS TANK INCOMING DIW SUPPLY AV3-1 (-161Y6) *)
	WY11605_11 AT  %MX11620.11 : BOOL; (*STN 3 PROCESS TANK INCOMING DIW SUPPLY AV3-1 (-161Y6) *)
	WY11605_12 AT  %MX11620.12 : BOOL; (*STN 3 PROCESS TANK INCOMING DIW SUPPLY AV3-1 (-161Y6) *)
	WY11605_13 AT  %MX11620.13 : BOOL; (*STN 3 PROCESS TANK INCOMING DIW SUPPLY AV3-1 (-161Y6) *)
	WY11605_14 AT  %MX11620.14 : BOOL; (*STN 3 PROCESS TANK INCOMING DIW SUPPLY AV3-1 (-161Y6) *)
	WY11605_15 AT  %MX11620.15 : BOOL; (*STN 3 PROCESS TANK INCOMING DIW SUPPLY AV3-1 (-161Y6) *)
	WY11605_16 AT  %MX11620.16 : BOOL; (*STN 3 PROCESS TANK INCOMING DIW SUPPLY AV3-1 (-161Y6) *)
	WY11605_17 AT  %MX11620.17 : BOOL; (*STN 3 PROCESS TANK INCOMING DIW SUPPLY AV3-1 (-161Y6) *)
	WY11605_18 AT  %MX11620.18 : BOOL; (*STN 3 PROCESS TANK INCOMING DIW SUPPLY AV3-1 (-161Y6) *)
	WY11605_19 AT  %MX11620.19 : BOOL; (*STN 3 PROCESS TANK INCOMING DIW SUPPLY AV3-1 (-161Y6) *)
	WY11605_20 AT  %MX11620.20 : BOOL; (*STN 3 PROCESS TANK INCOMING DIW SUPPLY AV3-1 (-161Y6) *)
	WY11605_21 AT  %MX11620.21 : BOOL; (*STN 3 PROCESS TANK INCOMING DIW SUPPLY AV3-1 (-161Y6) *)
	WY11605_22 AT  %MX11620.22 : BOOL; (*STN 3 PROCESS TANK INCOMING DIW SUPPLY AV3-1 (-161Y6) *)
	WY11605_23 AT  %MX11620.23 : BOOL; (*STN 3 PROCESS TANK INCOMING DIW SUPPLY AV3-1 (-161Y6) *)
	WY11605_24 AT  %MX11620.24 : BOOL; (*STN 3 PROCESS TANK INCOMING DIW SUPPLY AV3-1 (-161Y6) *)
	WY11605_25 AT  %MX11620.25 : BOOL; (*STN 3 PROCESS TANK INCOMING DIW SUPPLY AV3-1 (-161Y6) *)
	WY11605_26 AT  %MX11620.26 : BOOL; (*STN 3 PROCESS TANK INCOMING DIW SUPPLY AV3-1 (-161Y6) *)
	WY11605_27 AT  %MX11620.27 : BOOL; (*STN 3 PROCESS TANK INCOMING DIW SUPPLY AV3-1 (-161Y6) *)
	WY11605_28 AT  %MX11620.28 : BOOL; (*STN 3 PROCESS TANK INCOMING DIW SUPPLY AV3-1 (-161Y6) *)
	WY11605_29 AT  %MX11620.29 : BOOL; (*STN 3 PROCESS TANK INCOMING DIW SUPPLY AV3-1 (-161Y6) *)
	WY11605_30 AT  %MX11620.30 : BOOL; (*STN 3 PROCESS TANK INCOMING DIW SUPPLY AV3-1 (-161Y6) *)
	WY11605_31 AT  %MX11620.31 : BOOL; (*STN 3 PROCESS TANK INCOMING DIW SUPPLY AV3-1 (-161Y6) *)

	WY11606_00 AT  %MX11624.0 : BOOL; (*STN 4 PROCESS TANK CDA DISCHARGE AV4-1 (-161Y7) *)
	WY11606_01 AT  %MX11624.1 : BOOL; (*STN 4 PROCESS TANK CDA DISCHARGE AV4-1 (-161Y7) *)
	WY11606_02 AT  %MX11624.2 : BOOL; (*STN 4 PROCESS TANK CDA DISCHARGE AV4-1 (-161Y7) *)
	WY11606_03 AT  %MX11624.3 : BOOL; (*STN 4 PROCESS TANK CDA DISCHARGE AV4-1 (-161Y7) *)
	WY11606_04 AT  %MX11624.4 : BOOL; (*STN 4 PROCESS TANK CDA DISCHARGE AV4-1 (-161Y7) *)
	WY11606_05 AT  %MX11624.5 : BOOL; (*STN 4 PROCESS TANK CDA DISCHARGE AV4-1 (-161Y7) *)
	WY11606_06 AT  %MX11624.6 : BOOL; (*STN 4 PROCESS TANK CDA DISCHARGE AV4-1 (-161Y7) *)
	WY11606_07 AT  %MX11624.7 : BOOL; (*STN 4 PROCESS TANK CDA DISCHARGE AV4-1 (-161Y7) *)
	WY11606_08 AT  %MX11624.8 : BOOL; (*STN 4 PROCESS TANK CDA DISCHARGE AV4-1 (-161Y7) *)
	WY11606_09 AT  %MX11624.9 : BOOL; (*STN 4 PROCESS TANK CDA DISCHARGE AV4-1 (-161Y7) *)
	WY11606_10 AT  %MX11624.10 : BOOL; (*STN 4 PROCESS TANK CDA DISCHARGE AV4-1 (-161Y7) *)
	WY11606_11 AT  %MX11624.11 : BOOL; (*STN 4 PROCESS TANK CDA DISCHARGE AV4-1 (-161Y7) *)
	WY11606_12 AT  %MX11624.12 : BOOL; (*STN 4 PROCESS TANK CDA DISCHARGE AV4-1 (-161Y7) *)
	WY11606_13 AT  %MX11624.13 : BOOL; (*STN 4 PROCESS TANK CDA DISCHARGE AV4-1 (-161Y7) *)
	WY11606_14 AT  %MX11624.14 : BOOL; (*STN 4 PROCESS TANK CDA DISCHARGE AV4-1 (-161Y7) *)
	WY11606_15 AT  %MX11624.15 : BOOL; (*STN 4 PROCESS TANK CDA DISCHARGE AV4-1 (-161Y7) *)
	WY11606_16 AT  %MX11624.16 : BOOL; (*STN 4 PROCESS TANK CDA DISCHARGE AV4-1 (-161Y7) *)
	WY11606_17 AT  %MX11624.17 : BOOL; (*STN 4 PROCESS TANK CDA DISCHARGE AV4-1 (-161Y7) *)
	WY11606_18 AT  %MX11624.18 : BOOL; (*STN 4 PROCESS TANK CDA DISCHARGE AV4-1 (-161Y7) *)
	WY11606_19 AT  %MX11624.19 : BOOL; (*STN 4 PROCESS TANK CDA DISCHARGE AV4-1 (-161Y7) *)
	WY11606_20 AT  %MX11624.20 : BOOL; (*STN 4 PROCESS TANK CDA DISCHARGE AV4-1 (-161Y7) *)
	WY11606_21 AT  %MX11624.21 : BOOL; (*STN 4 PROCESS TANK CDA DISCHARGE AV4-1 (-161Y7) *)
	WY11606_22 AT  %MX11624.22 : BOOL; (*STN 4 PROCESS TANK CDA DISCHARGE AV4-1 (-161Y7) *)
	WY11606_23 AT  %MX11624.23 : BOOL; (*STN 4 PROCESS TANK CDA DISCHARGE AV4-1 (-161Y7) *)
	WY11606_24 AT  %MX11624.24 : BOOL; (*STN 4 PROCESS TANK CDA DISCHARGE AV4-1 (-161Y7) *)
	WY11606_25 AT  %MX11624.25 : BOOL; (*STN 4 PROCESS TANK CDA DISCHARGE AV4-1 (-161Y7) *)
	WY11606_26 AT  %MX11624.26 : BOOL; (*STN 4 PROCESS TANK CDA DISCHARGE AV4-1 (-161Y7) *)
	WY11606_27 AT  %MX11624.27 : BOOL; (*STN 4 PROCESS TANK CDA DISCHARGE AV4-1 (-161Y7) *)
	WY11606_28 AT  %MX11624.28 : BOOL; (*STN 4 PROCESS TANK CDA DISCHARGE AV4-1 (-161Y7) *)
	WY11606_29 AT  %MX11624.29 : BOOL; (*STN 4 PROCESS TANK CDA DISCHARGE AV4-1 (-161Y7) *)
	WY11606_30 AT  %MX11624.30 : BOOL; (*STN 4 PROCESS TANK CDA DISCHARGE AV4-1 (-161Y7) *)
	WY11606_31 AT  %MX11624.31 : BOOL; (*STN 4 PROCESS TANK CDA DISCHARGE AV4-1 (-161Y7) *)

	WY11607_00 AT  %MX11628.0 : BOOL; (*STN 4 PROCESS TANK CDA DISCHARGE AV4-2 (-161Y8) *)
	WY11607_01 AT  %MX11628.1 : BOOL; (*STN 4 PROCESS TANK CDA DISCHARGE AV4-2 (-161Y8) *)
	WY11607_02 AT  %MX11628.2 : BOOL; (*STN 4 PROCESS TANK CDA DISCHARGE AV4-2 (-161Y8) *)
	WY11607_03 AT  %MX11628.3 : BOOL; (*STN 4 PROCESS TANK CDA DISCHARGE AV4-2 (-161Y8) *)
	WY11607_04 AT  %MX11628.4 : BOOL; (*STN 4 PROCESS TANK CDA DISCHARGE AV4-2 (-161Y8) *)
	WY11607_05 AT  %MX11628.5 : BOOL; (*STN 4 PROCESS TANK CDA DISCHARGE AV4-2 (-161Y8) *)
	WY11607_06 AT  %MX11628.6 : BOOL; (*STN 4 PROCESS TANK CDA DISCHARGE AV4-2 (-161Y8) *)
	WY11607_07 AT  %MX11628.7 : BOOL; (*STN 4 PROCESS TANK CDA DISCHARGE AV4-2 (-161Y8) *)
	WY11607_08 AT  %MX11628.8 : BOOL; (*STN 4 PROCESS TANK CDA DISCHARGE AV4-2 (-161Y8) *)
	WY11607_09 AT  %MX11628.9 : BOOL; (*STN 4 PROCESS TANK CDA DISCHARGE AV4-2 (-161Y8) *)
	WY11607_10 AT  %MX11628.10 : BOOL; (*STN 4 PROCESS TANK CDA DISCHARGE AV4-2 (-161Y8) *)
	WY11607_11 AT  %MX11628.11 : BOOL; (*STN 4 PROCESS TANK CDA DISCHARGE AV4-2 (-161Y8) *)
	WY11607_12 AT  %MX11628.12 : BOOL; (*STN 4 PROCESS TANK CDA DISCHARGE AV4-2 (-161Y8) *)
	WY11607_13 AT  %MX11628.13 : BOOL; (*STN 4 PROCESS TANK CDA DISCHARGE AV4-2 (-161Y8) *)
	WY11607_14 AT  %MX11628.14 : BOOL; (*STN 4 PROCESS TANK CDA DISCHARGE AV4-2 (-161Y8) *)
	WY11607_15 AT  %MX11628.15 : BOOL; (*STN 4 PROCESS TANK CDA DISCHARGE AV4-2 (-161Y8) *)
	WY11607_16 AT  %MX11628.16 : BOOL; (*STN 4 PROCESS TANK CDA DISCHARGE AV4-2 (-161Y8) *)
	WY11607_17 AT  %MX11628.17 : BOOL; (*STN 4 PROCESS TANK CDA DISCHARGE AV4-2 (-161Y8) *)
	WY11607_18 AT  %MX11628.18 : BOOL; (*STN 4 PROCESS TANK CDA DISCHARGE AV4-2 (-161Y8) *)
	WY11607_19 AT  %MX11628.19 : BOOL; (*STN 4 PROCESS TANK CDA DISCHARGE AV4-2 (-161Y8) *)
	WY11607_20 AT  %MX11628.20 : BOOL; (*STN 4 PROCESS TANK CDA DISCHARGE AV4-2 (-161Y8) *)
	WY11607_21 AT  %MX11628.21 : BOOL; (*STN 4 PROCESS TANK CDA DISCHARGE AV4-2 (-161Y8) *)
	WY11607_22 AT  %MX11628.22 : BOOL; (*STN 4 PROCESS TANK CDA DISCHARGE AV4-2 (-161Y8) *)
	WY11607_23 AT  %MX11628.23 : BOOL; (*STN 4 PROCESS TANK CDA DISCHARGE AV4-2 (-161Y8) *)
	WY11607_24 AT  %MX11628.24 : BOOL; (*STN 4 PROCESS TANK CDA DISCHARGE AV4-2 (-161Y8) *)
	WY11607_25 AT  %MX11628.25 : BOOL; (*STN 4 PROCESS TANK CDA DISCHARGE AV4-2 (-161Y8) *)
	WY11607_26 AT  %MX11628.26 : BOOL; (*STN 4 PROCESS TANK CDA DISCHARGE AV4-2 (-161Y8) *)
	WY11607_27 AT  %MX11628.27 : BOOL; (*STN 4 PROCESS TANK CDA DISCHARGE AV4-2 (-161Y8) *)
	WY11607_28 AT  %MX11628.28 : BOOL; (*STN 4 PROCESS TANK CDA DISCHARGE AV4-2 (-161Y8) *)
	WY11607_29 AT  %MX11628.29 : BOOL; (*STN 4 PROCESS TANK CDA DISCHARGE AV4-2 (-161Y8) *)
	WY11607_30 AT  %MX11628.30 : BOOL; (*STN 4 PROCESS TANK CDA DISCHARGE AV4-2 (-161Y8) *)
	WY11607_31 AT  %MX11628.31 : BOOL; (*STN 4 PROCESS TANK CDA DISCHARGE AV4-2 (-161Y8) *)

	WY11608_00 AT  %MX11632.0 : BOOL; (*STN 5 PROCESS TANK VACUUM SUCTION AV5-1 (-161Y9) *)
	WY11608_01 AT  %MX11632.1 : BOOL; (*STN 5 PROCESS TANK VACUUM SUCTION AV5-1 (-161Y9) *)
	WY11608_02 AT  %MX11632.2 : BOOL; (*STN 5 PROCESS TANK VACUUM SUCTION AV5-1 (-161Y9) *)
	WY11608_03 AT  %MX11632.3 : BOOL; (*STN 5 PROCESS TANK VACUUM SUCTION AV5-1 (-161Y9) *)
	WY11608_04 AT  %MX11632.4 : BOOL; (*STN 5 PROCESS TANK VACUUM SUCTION AV5-1 (-161Y9) *)
	WY11608_05 AT  %MX11632.5 : BOOL; (*STN 5 PROCESS TANK VACUUM SUCTION AV5-1 (-161Y9) *)
	WY11608_06 AT  %MX11632.6 : BOOL; (*STN 5 PROCESS TANK VACUUM SUCTION AV5-1 (-161Y9) *)
	WY11608_07 AT  %MX11632.7 : BOOL; (*STN 5 PROCESS TANK VACUUM SUCTION AV5-1 (-161Y9) *)
	WY11608_08 AT  %MX11632.8 : BOOL; (*STN 5 PROCESS TANK VACUUM SUCTION AV5-1 (-161Y9) *)
	WY11608_09 AT  %MX11632.9 : BOOL; (*STN 5 PROCESS TANK VACUUM SUCTION AV5-1 (-161Y9) *)
	WY11608_10 AT  %MX11632.10 : BOOL; (*STN 5 PROCESS TANK VACUUM SUCTION AV5-1 (-161Y9) *)
	WY11608_11 AT  %MX11632.11 : BOOL; (*STN 5 PROCESS TANK VACUUM SUCTION AV5-1 (-161Y9) *)
	WY11608_12 AT  %MX11632.12 : BOOL; (*STN 5 PROCESS TANK VACUUM SUCTION AV5-1 (-161Y9) *)
	WY11608_13 AT  %MX11632.13 : BOOL; (*STN 5 PROCESS TANK VACUUM SUCTION AV5-1 (-161Y9) *)
	WY11608_14 AT  %MX11632.14 : BOOL; (*STN 5 PROCESS TANK VACUUM SUCTION AV5-1 (-161Y9) *)
	WY11608_15 AT  %MX11632.15 : BOOL; (*STN 5 PROCESS TANK VACUUM SUCTION AV5-1 (-161Y9) *)
	WY11608_16 AT  %MX11632.16 : BOOL; (*STN 5 PROCESS TANK VACUUM SUCTION AV5-1 (-161Y9) *)
	WY11608_17 AT  %MX11632.17 : BOOL; (*STN 5 PROCESS TANK VACUUM SUCTION AV5-1 (-161Y9) *)
	WY11608_18 AT  %MX11632.18 : BOOL; (*STN 5 PROCESS TANK VACUUM SUCTION AV5-1 (-161Y9) *)
	WY11608_19 AT  %MX11632.19 : BOOL; (*STN 5 PROCESS TANK VACUUM SUCTION AV5-1 (-161Y9) *)
	WY11608_20 AT  %MX11632.20 : BOOL; (*STN 5 PROCESS TANK VACUUM SUCTION AV5-1 (-161Y9) *)
	WY11608_21 AT  %MX11632.21 : BOOL; (*STN 5 PROCESS TANK VACUUM SUCTION AV5-1 (-161Y9) *)
	WY11608_22 AT  %MX11632.22 : BOOL; (*STN 5 PROCESS TANK VACUUM SUCTION AV5-1 (-161Y9) *)
	WY11608_23 AT  %MX11632.23 : BOOL; (*STN 5 PROCESS TANK VACUUM SUCTION AV5-1 (-161Y9) *)
	WY11608_24 AT  %MX11632.24 : BOOL; (*STN 5 PROCESS TANK VACUUM SUCTION AV5-1 (-161Y9) *)
	WY11608_25 AT  %MX11632.25 : BOOL; (*STN 5 PROCESS TANK VACUUM SUCTION AV5-1 (-161Y9) *)
	WY11608_26 AT  %MX11632.26 : BOOL; (*STN 5 PROCESS TANK VACUUM SUCTION AV5-1 (-161Y9) *)
	WY11608_27 AT  %MX11632.27 : BOOL; (*STN 5 PROCESS TANK VACUUM SUCTION AV5-1 (-161Y9) *)
	WY11608_28 AT  %MX11632.28 : BOOL; (*STN 5 PROCESS TANK VACUUM SUCTION AV5-1 (-161Y9) *)
	WY11608_29 AT  %MX11632.29 : BOOL; (*STN 5 PROCESS TANK VACUUM SUCTION AV5-1 (-161Y9) *)
	WY11608_30 AT  %MX11632.30 : BOOL; (*STN 5 PROCESS TANK VACUUM SUCTION AV5-1 (-161Y9) *)
	WY11608_31 AT  %MX11632.31 : BOOL; (*STN 5 PROCESS TANK VACUUM SUCTION AV5-1 (-161Y9) *)

